REGION Network 41: RO-2 A AUTO FLUSING VALVE AGLV-401 CLOSE COMMOND FAIL
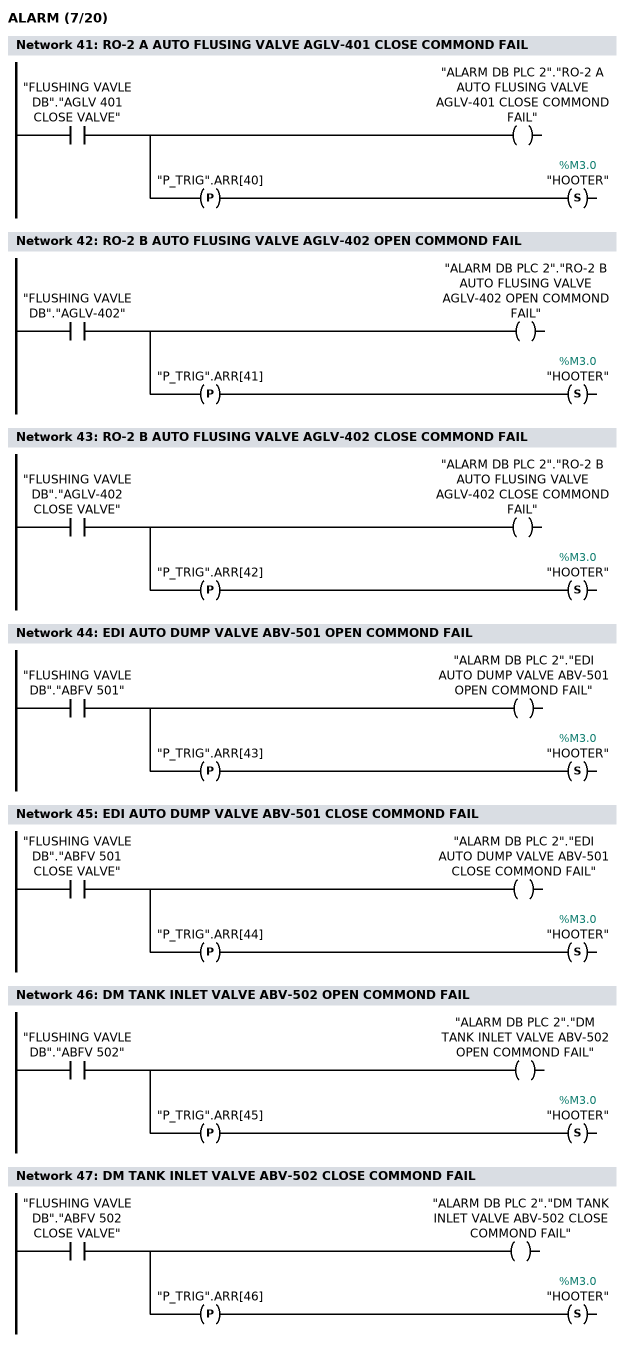
   RUNG wire#powerrail
      Contact( "FLUSHING VAVLE DB"."AGLV 401 CLOSE VALVE" )
      wire#w1
      Coil( "ALARM DB PLC 2"."RO-2 A AUTO FLUSING VALVE AGLV-401 CLOSE COMMOND FAIL" )
   END_RUNG
   RUNG wire#w1
      P_Trig( "P_TRIG".ARR[40] )
      S_Coil( "HOOTER" )
   END_RUNG
   // the same network as SCL:
   "ALARM DB PLC 2"."RO-2 A AUTO FLUSING VALVE AGLV-401 CLOSE COMMOND FAIL" := "FLUSHING VAVLE DB"."AGLV 401 CLOSE VALVE";
   #_w1 := "FLUSHING VAVLE DB"."AGLV 401 CLOSE VALVE" AND NOT "P_TRIG".ARR[40];   // rising edge
   "P_TRIG".ARR[40] := "FLUSHING VAVLE DB"."AGLV 401 CLOSE VALVE";
   IF #_w1 THEN "HOOTER" := TRUE; END_IF;
END_REGION

REGION Network 42: RO-2 B AUTO FLUSING VALVE AGLV-402 OPEN COMMOND FAIL
   RUNG wire#powerrail
      Contact( "FLUSHING VAVLE DB"."AGLV-402" )
      wire#w1
      Coil( "ALARM DB PLC 2"."RO-2 B AUTO FLUSING VALVE AGLV-402 OPEN COMMOND FAIL" )
   END_RUNG
   RUNG wire#w1
      P_Trig( "P_TRIG".ARR[41] )
      S_Coil( "HOOTER" )
   END_RUNG
   // the same network as SCL:
   "ALARM DB PLC 2"."RO-2 B AUTO FLUSING VALVE AGLV-402 OPEN COMMOND FAIL" := "FLUSHING VAVLE DB"."AGLV-402";
   #_w1 := "FLUSHING VAVLE DB"."AGLV-402" AND NOT "P_TRIG".ARR[41];   // rising edge
   "P_TRIG".ARR[41] := "FLUSHING VAVLE DB"."AGLV-402";
   IF #_w1 THEN "HOOTER" := TRUE; END_IF;
END_REGION

REGION Network 43: RO-2 B AUTO FLUSING VALVE AGLV-402 CLOSE COMMOND FAIL
   RUNG wire#powerrail
      Contact( "FLUSHING VAVLE DB"."AGLV-402 CLOSE VALVE" )
      wire#w1
      Coil( "ALARM DB PLC 2"."RO-2 B AUTO FLUSING VALVE AGLV-402 CLOSE COMMOND FAIL" )
   END_RUNG
   RUNG wire#w1
      P_Trig( "P_TRIG".ARR[42] )
      S_Coil( "HOOTER" )
   END_RUNG
   // the same network as SCL:
   "ALARM DB PLC 2"."RO-2 B AUTO FLUSING VALVE AGLV-402 CLOSE COMMOND FAIL" := "FLUSHING VAVLE DB"."AGLV-402 CLOSE VALVE";
   #_w1 := "FLUSHING VAVLE DB"."AGLV-402 CLOSE VALVE" AND NOT "P_TRIG".ARR[42];   // rising edge
   "P_TRIG".ARR[42] := "FLUSHING VAVLE DB"."AGLV-402 CLOSE VALVE";
   IF #_w1 THEN "HOOTER" := TRUE; END_IF;
END_REGION

REGION Network 44: EDI AUTO DUMP VALVE ABV-501 OPEN COMMOND FAIL
   RUNG wire#powerrail
      Contact( "FLUSHING VAVLE DB"."ABFV 501" )
      wire#w1
      Coil( "ALARM DB PLC 2"."EDI AUTO DUMP VALVE ABV-501 OPEN COMMOND FAIL" )
   END_RUNG
   RUNG wire#w1
      P_Trig( "P_TRIG".ARR[43] )
      S_Coil( "HOOTER" )
   END_RUNG
   // the same network as SCL:
   "ALARM DB PLC 2"."EDI AUTO DUMP VALVE ABV-501 OPEN COMMOND FAIL" := "FLUSHING VAVLE DB"."ABFV 501";
   #_w1 := "FLUSHING VAVLE DB"."ABFV 501" AND NOT "P_TRIG".ARR[43];   // rising edge
   "P_TRIG".ARR[43] := "FLUSHING VAVLE DB"."ABFV 501";
   IF #_w1 THEN "HOOTER" := TRUE; END_IF;
END_REGION

REGION Network 45: EDI AUTO DUMP VALVE ABV-501 CLOSE COMMOND FAIL
   RUNG wire#powerrail
      Contact( "FLUSHING VAVLE DB"."ABFV 501 CLOSE VALVE" )
      wire#w1
      Coil( "ALARM DB PLC 2"."EDI AUTO DUMP VALVE ABV-501 CLOSE COMMOND FAIL" )
   END_RUNG
   RUNG wire#w1
      P_Trig( "P_TRIG".ARR[44] )
      S_Coil( "HOOTER" )
   END_RUNG
   // the same network as SCL:
   "ALARM DB PLC 2"."EDI AUTO DUMP VALVE ABV-501 CLOSE COMMOND FAIL" := "FLUSHING VAVLE DB"."ABFV 501 CLOSE VALVE";
   #_w1 := "FLUSHING VAVLE DB"."ABFV 501 CLOSE VALVE" AND NOT "P_TRIG".ARR[44];   // rising edge
   "P_TRIG".ARR[44] := "FLUSHING VAVLE DB"."ABFV 501 CLOSE VALVE";
   IF #_w1 THEN "HOOTER" := TRUE; END_IF;
END_REGION

REGION Network 46: DM TANK INLET VALVE ABV-502 OPEN COMMOND FAIL
   RUNG wire#powerrail
      Contact( "FLUSHING VAVLE DB"."ABFV 502" )
      wire#w1
      Coil( "ALARM DB PLC 2"."DM TANK INLET VALVE ABV-502 OPEN COMMOND FAIL" )
   END_RUNG
   RUNG wire#w1
      P_Trig( "P_TRIG".ARR[45] )
      S_Coil( "HOOTER" )
   END_RUNG
   // the same network as SCL:
   "ALARM DB PLC 2"."DM TANK INLET VALVE ABV-502 OPEN COMMOND FAIL" := "FLUSHING VAVLE DB"."ABFV 502";
   #_w1 := "FLUSHING VAVLE DB"."ABFV 502" AND NOT "P_TRIG".ARR[45];   // rising edge
   "P_TRIG".ARR[45] := "FLUSHING VAVLE DB"."ABFV 502";
   IF #_w1 THEN "HOOTER" := TRUE; END_IF;
END_REGION

REGION Network 47: DM TANK INLET VALVE ABV-502 CLOSE COMMOND FAIL
   RUNG wire#powerrail
      Contact( "FLUSHING VAVLE DB"."ABFV 502 CLOSE VALVE" )
      wire#w1
      Coil( "ALARM DB PLC 2"."DM TANK INLET VALVE ABV-502 CLOSE COMMOND FAIL" )
   END_RUNG
   RUNG wire#w1
      P_Trig( "P_TRIG".ARR[46] )
      S_Coil( "HOOTER" )
   END_RUNG
   // the same network as SCL:
   "ALARM DB PLC 2"."DM TANK INLET VALVE ABV-502 CLOSE COMMOND FAIL" := "FLUSHING VAVLE DB"."ABFV 502 CLOSE VALVE";
   #_w1 := "FLUSHING VAVLE DB"."ABFV 502 CLOSE VALVE" AND NOT "P_TRIG".ARR[46];   // rising edge
   "P_TRIG".ARR[46] := "FLUSHING VAVLE DB"."ABFV 502 CLOSE VALVE";
   IF #_w1 THEN "HOOTER" := TRUE; END_IF;
END_REGION

REGION Network 48: RO-02 FEED TANK LEVEL ( LT-401)- LOW LOW
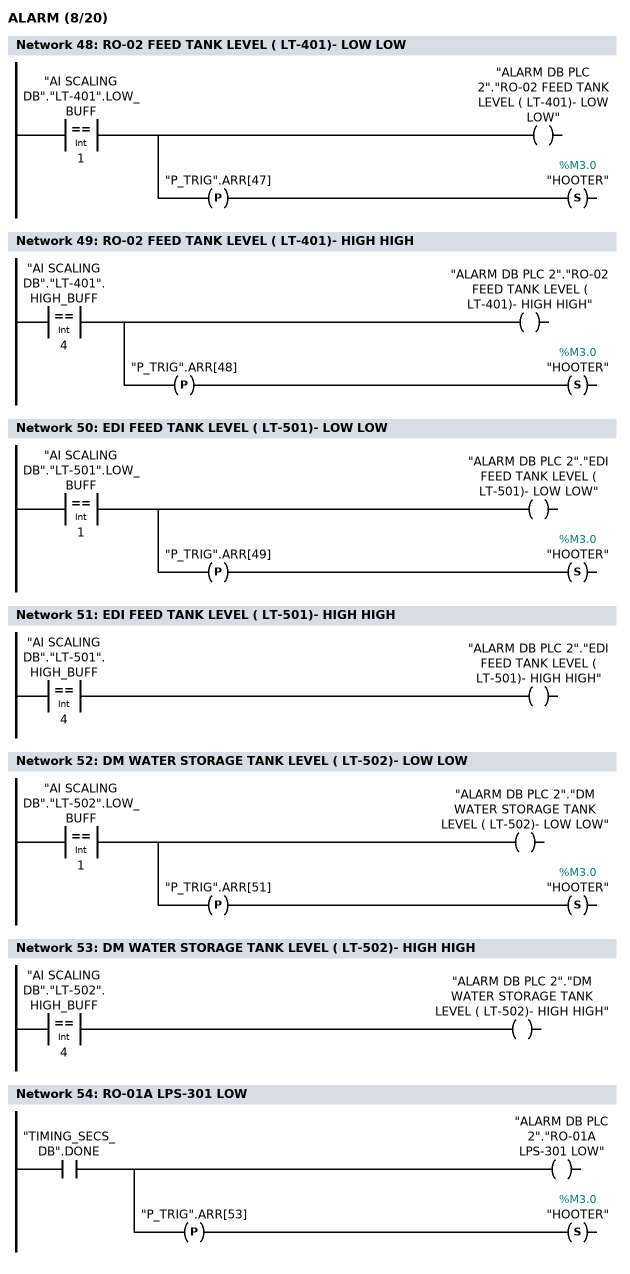
   RUNG wire#powerrail
      { S7_Templates := "SrcType := Int" } EQ_Contact(in1 := "AI SCALING DB"."LT-401".LOW_BUFF, in2 := 1)
      wire#w1
      Coil( "ALARM DB PLC 2"."RO-02 FEED TANK LEVEL ( LT-401)- LOW LOW" )
   END_RUNG
   RUNG wire#w1
      P_Trig( "P_TRIG".ARR[47] )
      S_Coil( "HOOTER" )
   END_RUNG
   // the same network as SCL:
   "ALARM DB PLC 2"."RO-02 FEED TANK LEVEL ( LT-401)- LOW LOW" := "AI SCALING DB"."LT-401".LOW_BUFF = 1;
   #_w1 := "ALARM DB PLC 2"."RO-02 FEED TANK LEVEL ( LT-401)- LOW LOW" AND NOT "P_TRIG".ARR[47];   // rising edge
   "P_TRIG".ARR[47] := "ALARM DB PLC 2"."RO-02 FEED TANK LEVEL ( LT-401)- LOW LOW";
   IF #_w1 THEN "HOOTER" := TRUE; END_IF;
END_REGION

REGION Network 49: RO-02 FEED TANK LEVEL ( LT-401)- HIGH HIGH
   RUNG wire#powerrail
      { S7_Templates := "SrcType := Int" } EQ_Contact(in1 := "AI SCALING DB"."LT-401".HIGH_BUFF, in2 := 4)
      wire#w1
      Coil( "ALARM DB PLC 2"."RO-02 FEED TANK LEVEL ( LT-401)- HIGH HIGH" )
   END_RUNG
   RUNG wire#w1
      P_Trig( "P_TRIG".ARR[48] )
      S_Coil( "HOOTER" )
   END_RUNG
   // the same network as SCL:
   "ALARM DB PLC 2"."RO-02 FEED TANK LEVEL ( LT-401)- HIGH HIGH" := "AI SCALING DB"."LT-401".HIGH_BUFF = 4;
   #_w1 := "ALARM DB PLC 2"."RO-02 FEED TANK LEVEL ( LT-401)- HIGH HIGH" AND NOT "P_TRIG".ARR[48];   // rising edge
   "P_TRIG".ARR[48] := "ALARM DB PLC 2"."RO-02 FEED TANK LEVEL ( LT-401)- HIGH HIGH";
   IF #_w1 THEN "HOOTER" := TRUE; END_IF;
END_REGION

REGION Network 50: EDI FEED TANK LEVEL ( LT-501)- LOW LOW
   RUNG wire#powerrail
      { S7_Templates := "SrcType := Int" } EQ_Contact(in1 := "AI SCALING DB"."LT-501".LOW_BUFF, in2 := 1)
      wire#w1
      Coil( "ALARM DB PLC 2"."EDI FEED TANK LEVEL ( LT-501)- LOW LOW" )
   END_RUNG
   RUNG wire#w1
      P_Trig( "P_TRIG".ARR[49] )
      S_Coil( "HOOTER" )
   END_RUNG
   // the same network as SCL:
   "ALARM DB PLC 2"."EDI FEED TANK LEVEL ( LT-501)- LOW LOW" := "AI SCALING DB"."LT-501".LOW_BUFF = 1;
   #_w1 := "ALARM DB PLC 2"."EDI FEED TANK LEVEL ( LT-501)- LOW LOW" AND NOT "P_TRIG".ARR[49];   // rising edge
   "P_TRIG".ARR[49] := "ALARM DB PLC 2"."EDI FEED TANK LEVEL ( LT-501)- LOW LOW";
   IF #_w1 THEN "HOOTER" := TRUE; END_IF;
END_REGION

REGION Network 51: EDI FEED TANK LEVEL ( LT-501)- HIGH HIGH
   RUNG wire#powerrail
      { S7_Templates := "SrcType := Int" } EQ_Contact(in1 := "AI SCALING DB"."LT-501".HIGH_BUFF, in2 := 4)
      Coil( "ALARM DB PLC 2"."EDI FEED TANK LEVEL ( LT-501)- HIGH HIGH" )
   END_RUNG
   // the same network as SCL:
   "ALARM DB PLC 2"."EDI FEED TANK LEVEL ( LT-501)- HIGH HIGH" := "AI SCALING DB"."LT-501".HIGH_BUFF = 4;
END_REGION

REGION Network 52: DM WATER STORAGE TANK LEVEL ( LT-502)- LOW LOW
   RUNG wire#powerrail
      { S7_Templates := "SrcType := Int" } EQ_Contact(in1 := "AI SCALING DB"."LT-502".LOW_BUFF, in2 := 1)
      wire#w1
      Coil( "ALARM DB PLC 2"."DM WATER STORAGE TANK  LEVEL ( LT-502)- LOW LOW" )
   END_RUNG
   RUNG wire#w1
      P_Trig( "P_TRIG".ARR[51] )
      S_Coil( "HOOTER" )
   END_RUNG
   // the same network as SCL:
   "ALARM DB PLC 2"."DM WATER STORAGE TANK  LEVEL ( LT-502)- LOW LOW" := "AI SCALING DB"."LT-502".LOW_BUFF = 1;
   #_w1 := "ALARM DB PLC 2"."DM WATER STORAGE TANK  LEVEL ( LT-502)- LOW LOW" AND NOT "P_TRIG".ARR[51];   // rising edge
   "P_TRIG".ARR[51] := "ALARM DB PLC 2"."DM WATER STORAGE TANK  LEVEL ( LT-502)- LOW LOW";
   IF #_w1 THEN "HOOTER" := TRUE; END_IF;
END_REGION

REGION Network 53: DM WATER STORAGE TANK LEVEL ( LT-502)- HIGH HIGH
   RUNG wire#powerrail
      { S7_Templates := "SrcType := Int" } EQ_Contact(in1 := "AI SCALING DB"."LT-502".HIGH_BUFF, in2 := 4)
      Coil( "ALARM DB PLC 2"."DM WATER STORAGE TANK LEVEL ( LT-502)- HIGH HIGH" )
   END_RUNG
   // the same network as SCL:
   "ALARM DB PLC 2"."DM WATER STORAGE TANK LEVEL ( LT-502)- HIGH HIGH" := "AI SCALING DB"."LT-502".HIGH_BUFF = 4;
END_REGION

REGION Network 54: RO-01A LPS-301 LOW
   RUNG wire#powerrail
      Contact( "TIMING_SECS_DB".DONE )
      wire#w1
      Coil( "ALARM DB PLC 2"."RO-01A LPS-301 LOW" )
   END_RUNG
   RUNG wire#w1
      P_Trig( "P_TRIG".ARR[53] )
      S_Coil( "HOOTER" )
   END_RUNG
   // the same network as SCL:
   "ALARM DB PLC 2"."RO-01A LPS-301 LOW" := "TIMING_SECS_DB".DONE;
   #_w1 := "TIMING_SECS_DB".DONE AND NOT "P_TRIG".ARR[53];   // rising edge
   "P_TRIG".ARR[53] := "TIMING_SECS_DB".DONE;
   IF #_w1 THEN "HOOTER" := TRUE; END_IF;
END_REGION

REGION Network 55: RO-01 B LPS-302 LOW
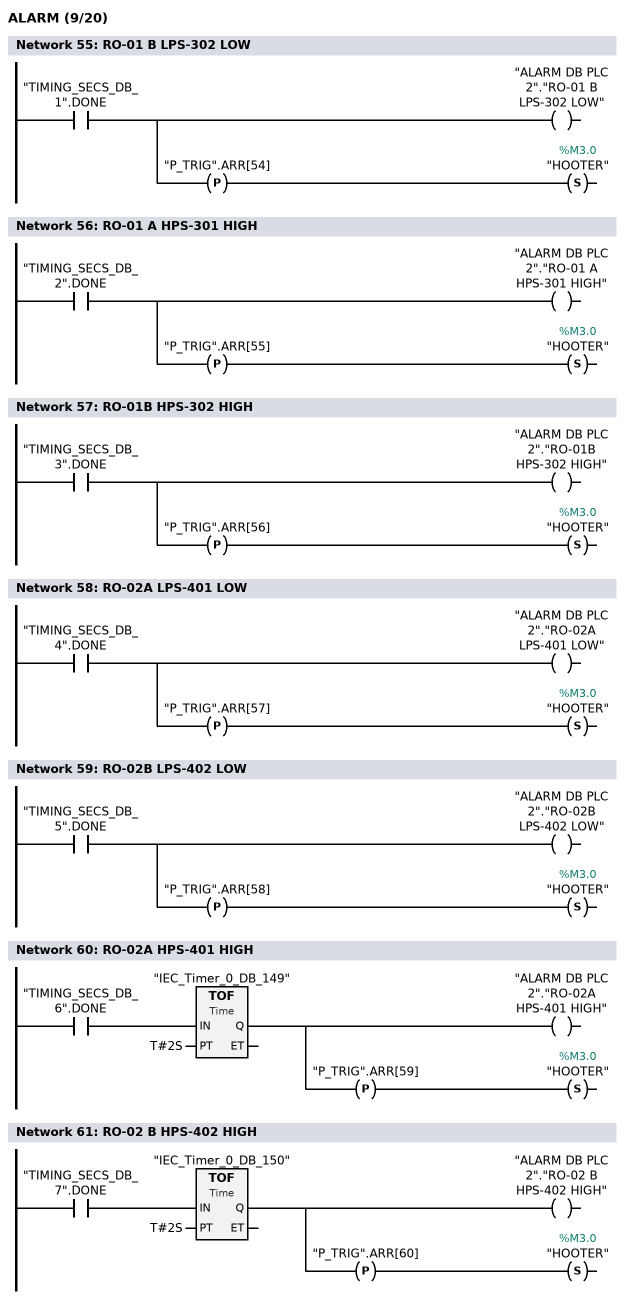
   RUNG wire#powerrail
      Contact( "TIMING_SECS_DB_1".DONE )
      wire#w1
      Coil( "ALARM DB PLC 2"."RO-01 B LPS-302 LOW" )
   END_RUNG
   RUNG wire#w1
      P_Trig( "P_TRIG".ARR[54] )
      S_Coil( "HOOTER" )
   END_RUNG
   // the same network as SCL:
   "ALARM DB PLC 2"."RO-01 B LPS-302 LOW" := "TIMING_SECS_DB_1".DONE;
   #_w1 := "TIMING_SECS_DB_1".DONE AND NOT "P_TRIG".ARR[54];   // rising edge
   "P_TRIG".ARR[54] := "TIMING_SECS_DB_1".DONE;
   IF #_w1 THEN "HOOTER" := TRUE; END_IF;
END_REGION

REGION Network 56: RO-01 A HPS-301 HIGH
   RUNG wire#powerrail
      Contact( "TIMING_SECS_DB_2".DONE )
      wire#w1
      Coil( "ALARM DB PLC 2"."RO-01 A HPS-301 HIGH" )
   END_RUNG
   RUNG wire#w1
      P_Trig( "P_TRIG".ARR[55] )
      S_Coil( "HOOTER" )
   END_RUNG
   // the same network as SCL:
   "ALARM DB PLC 2"."RO-01 A HPS-301 HIGH" := "TIMING_SECS_DB_2".DONE;
   #_w1 := "TIMING_SECS_DB_2".DONE AND NOT "P_TRIG".ARR[55];   // rising edge
   "P_TRIG".ARR[55] := "TIMING_SECS_DB_2".DONE;
   IF #_w1 THEN "HOOTER" := TRUE; END_IF;
END_REGION

REGION Network 57: RO-01B HPS-302 HIGH
   RUNG wire#powerrail
      Contact( "TIMING_SECS_DB_3".DONE )
      wire#w1
      Coil( "ALARM DB PLC 2"."RO-01B HPS-302 HIGH" )
   END_RUNG
   RUNG wire#w1
      P_Trig( "P_TRIG".ARR[56] )
      S_Coil( "HOOTER" )
   END_RUNG
   // the same network as SCL:
   "ALARM DB PLC 2"."RO-01B HPS-302 HIGH" := "TIMING_SECS_DB_3".DONE;
   #_w1 := "TIMING_SECS_DB_3".DONE AND NOT "P_TRIG".ARR[56];   // rising edge
   "P_TRIG".ARR[56] := "TIMING_SECS_DB_3".DONE;
   IF #_w1 THEN "HOOTER" := TRUE; END_IF;
END_REGION

REGION Network 58: RO-02A LPS-401 LOW
   RUNG wire#powerrail
      Contact( "TIMING_SECS_DB_4".DONE )
      wire#w1
      Coil( "ALARM DB PLC 2"."RO-02A LPS-401 LOW" )
   END_RUNG
   RUNG wire#w1
      P_Trig( "P_TRIG".ARR[57] )
      S_Coil( "HOOTER" )
   END_RUNG
   // the same network as SCL:
   "ALARM DB PLC 2"."RO-02A LPS-401 LOW" := "TIMING_SECS_DB_4".DONE;
   #_w1 := "TIMING_SECS_DB_4".DONE AND NOT "P_TRIG".ARR[57];   // rising edge
   "P_TRIG".ARR[57] := "TIMING_SECS_DB_4".DONE;
   IF #_w1 THEN "HOOTER" := TRUE; END_IF;
END_REGION

REGION Network 59: RO-02B LPS-402 LOW
   RUNG wire#powerrail
      Contact( "TIMING_SECS_DB_5".DONE )
      wire#w1
      Coil( "ALARM DB PLC 2"."RO-02B LPS-402 LOW" )
   END_RUNG
   RUNG wire#w1
      P_Trig( "P_TRIG".ARR[58] )
      S_Coil( "HOOTER" )
   END_RUNG
   // the same network as SCL:
   "ALARM DB PLC 2"."RO-02B LPS-402 LOW" := "TIMING_SECS_DB_5".DONE;
   #_w1 := "TIMING_SECS_DB_5".DONE AND NOT "P_TRIG".ARR[58];   // rising edge
   "P_TRIG".ARR[58] := "TIMING_SECS_DB_5".DONE;
   IF #_w1 THEN "HOOTER" := TRUE; END_IF;
END_REGION

REGION Network 60: RO-02A HPS-401 HIGH
   RUNG wire#powerrail
      Contact( "TIMING_SECS_DB_6".DONE )
      { S7_Templates := "time_type := Time" } "IEC_Timer_0_DB_149".TOF(pt := T#2S, et =>)
      wire#w1
      Coil( "ALARM DB PLC 2"."RO-02A HPS-401 HIGH" )
   END_RUNG
   RUNG wire#w1
      P_Trig( "P_TRIG".ARR[59] )
      S_Coil( "HOOTER" )
   END_RUNG
   // the same network as SCL:
   "IEC_Timer_0_DB_149".TOF(IN := "TIMING_SECS_DB_6".DONE, PT := T#2S);
   "ALARM DB PLC 2"."RO-02A HPS-401 HIGH" := "IEC_Timer_0_DB_149".Q;
   #_w1 := "IEC_Timer_0_DB_149".Q AND NOT "P_TRIG".ARR[59];   // rising edge
   "P_TRIG".ARR[59] := "IEC_Timer_0_DB_149".Q;
   IF #_w1 THEN "HOOTER" := TRUE; END_IF;
END_REGION

REGION Network 61: RO-02 B HPS-402 HIGH
   RUNG wire#powerrail
      Contact( "TIMING_SECS_DB_7".DONE )
      { S7_Templates := "time_type := Time" } "IEC_Timer_0_DB_150".TOF(pt := T#2S, et =>)
      wire#w1
      Coil( "ALARM DB PLC 2"."RO-02 B HPS-402 HIGH" )
   END_RUNG
   RUNG wire#w1
      P_Trig( "P_TRIG".ARR[60] )
      S_Coil( "HOOTER" )
   END_RUNG
   // the same network as SCL:
   "IEC_Timer_0_DB_150".TOF(IN := "TIMING_SECS_DB_7".DONE, PT := T#2S);
   "ALARM DB PLC 2"."RO-02 B HPS-402 HIGH" := "IEC_Timer_0_DB_150".Q;
   #_w1 := "IEC_Timer_0_DB_150".Q AND NOT "P_TRIG".ARR[60];   // rising edge
   "P_TRIG".ARR[60] := "IEC_Timer_0_DB_150".Q;
   IF #_w1 THEN "HOOTER" := TRUE; END_IF;
END_REGION

REGION Network 62: EDI-501A FEED PRESSURE PT-501 LOW
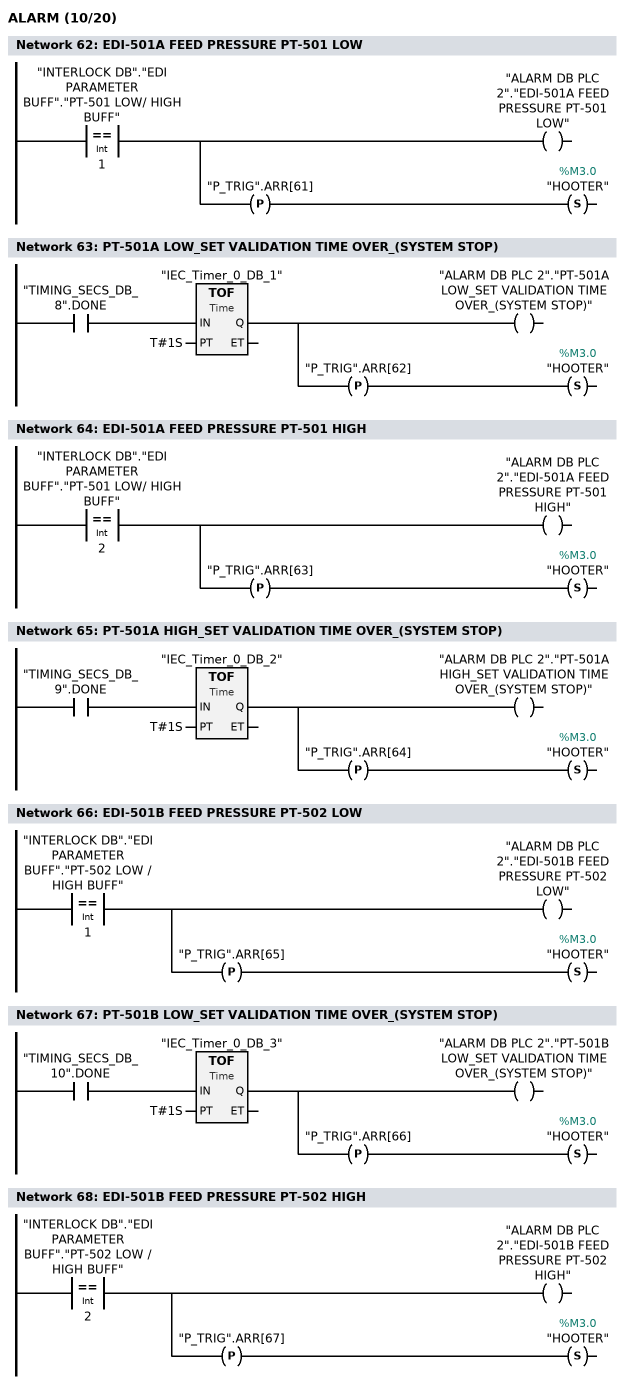
   RUNG wire#powerrail
      { S7_Templates := "SrcType := Int" } EQ_Contact(in1 := "INTERLOCK DB"."EDI PARAMETER BUFF"."PT-501 LOW/ HIGH BUFF", in2 := 1)
      wire#w1
      Coil( "ALARM DB PLC 2"."EDI-501A FEED PRESSURE PT-501 LOW" )
   END_RUNG
   RUNG wire#w1
      P_Trig( "P_TRIG".ARR[61] )
      S_Coil( "HOOTER" )
   END_RUNG
   // the same network as SCL:
   "ALARM DB PLC 2"."EDI-501A FEED PRESSURE PT-501 LOW" := "INTERLOCK DB"."EDI PARAMETER BUFF"."PT-501 LOW/ HIGH BUFF" = 1;
   #_w1 := "ALARM DB PLC 2"."EDI-501A FEED PRESSURE PT-501 LOW" AND NOT "P_TRIG".ARR[61];   // rising edge
   "P_TRIG".ARR[61] := "ALARM DB PLC 2"."EDI-501A FEED PRESSURE PT-501 LOW";
   IF #_w1 THEN "HOOTER" := TRUE; END_IF;
END_REGION

REGION Network 63: PT-501A LOW_SET VALIDATION TIME OVER_(SYSTEM STOP)
   RUNG wire#powerrail
      Contact( "TIMING_SECS_DB_8".DONE )
      { S7_Templates := "time_type := Time" } "IEC_Timer_0_DB_1".TOF(pt := T#1S, et =>)
      wire#w1
      Coil( "ALARM DB PLC 2"."PT-501A LOW_SET VALIDATION TIME OVER_(SYSTEM STOP)" )
   END_RUNG
   RUNG wire#w1
      P_Trig( "P_TRIG".ARR[62] )
      S_Coil( "HOOTER" )
   END_RUNG
   // the same network as SCL:
   "IEC_Timer_0_DB_1".TOF(IN := "TIMING_SECS_DB_8".DONE, PT := T#1S);
   "ALARM DB PLC 2"."PT-501A LOW_SET VALIDATION TIME OVER_(SYSTEM STOP)" := "IEC_Timer_0_DB_1".Q;
   #_w1 := "IEC_Timer_0_DB_1".Q AND NOT "P_TRIG".ARR[62];   // rising edge
   "P_TRIG".ARR[62] := "IEC_Timer_0_DB_1".Q;
   IF #_w1 THEN "HOOTER" := TRUE; END_IF;
END_REGION

REGION Network 64: EDI-501A FEED PRESSURE PT-501 HIGH
   RUNG wire#powerrail
      { S7_Templates := "SrcType := Int" } EQ_Contact(in1 := "INTERLOCK DB"."EDI PARAMETER BUFF"."PT-501 LOW/ HIGH BUFF", in2 := 2)
      wire#w1
      Coil( "ALARM DB PLC 2"."EDI-501A FEED PRESSURE PT-501 HIGH" )
   END_RUNG
   RUNG wire#w1
      P_Trig( "P_TRIG".ARR[63] )
      S_Coil( "HOOTER" )
   END_RUNG
   // the same network as SCL:
   "ALARM DB PLC 2"."EDI-501A FEED PRESSURE PT-501 HIGH" := "INTERLOCK DB"."EDI PARAMETER BUFF"."PT-501 LOW/ HIGH BUFF" = 2;
   #_w1 := "ALARM DB PLC 2"."EDI-501A FEED PRESSURE PT-501 HIGH" AND NOT "P_TRIG".ARR[63];   // rising edge
   "P_TRIG".ARR[63] := "ALARM DB PLC 2"."EDI-501A FEED PRESSURE PT-501 HIGH";
   IF #_w1 THEN "HOOTER" := TRUE; END_IF;
END_REGION

REGION Network 65: PT-501A HIGH_SET VALIDATION TIME OVER_(SYSTEM STOP)
   RUNG wire#powerrail
      Contact( "TIMING_SECS_DB_9".DONE )
      { S7_Templates := "time_type := Time" } "IEC_Timer_0_DB_2".TOF(pt := T#1S, et =>)
      wire#w1
      Coil( "ALARM DB PLC 2"."PT-501A HIGH_SET VALIDATION TIME OVER_(SYSTEM STOP)" )
   END_RUNG
   RUNG wire#w1
      P_Trig( "P_TRIG".ARR[64] )
      S_Coil( "HOOTER" )
   END_RUNG
   // the same network as SCL:
   "IEC_Timer_0_DB_2".TOF(IN := "TIMING_SECS_DB_9".DONE, PT := T#1S);
   "ALARM DB PLC 2"."PT-501A HIGH_SET VALIDATION TIME OVER_(SYSTEM STOP)" := "IEC_Timer_0_DB_2".Q;
   #_w1 := "IEC_Timer_0_DB_2".Q AND NOT "P_TRIG".ARR[64];   // rising edge
   "P_TRIG".ARR[64] := "IEC_Timer_0_DB_2".Q;
   IF #_w1 THEN "HOOTER" := TRUE; END_IF;
END_REGION

REGION Network 66: EDI-501B FEED PRESSURE PT-502 LOW
   RUNG wire#powerrail
      { S7_Templates := "SrcType := Int" } EQ_Contact(in1 := "INTERLOCK DB"."EDI PARAMETER BUFF"."PT-502 LOW / HIGH BUFF", in2 := 1)
      wire#w1
      Coil( "ALARM DB PLC 2"."EDI-501B FEED PRESSURE PT-502 LOW" )
   END_RUNG
   RUNG wire#w1
      P_Trig( "P_TRIG".ARR[65] )
      S_Coil( "HOOTER" )
   END_RUNG
   // the same network as SCL:
   "ALARM DB PLC 2"."EDI-501B FEED PRESSURE PT-502 LOW" := "INTERLOCK DB"."EDI PARAMETER BUFF"."PT-502 LOW / HIGH BUFF" = 1;
   #_w1 := "ALARM DB PLC 2"."EDI-501B FEED PRESSURE PT-502 LOW" AND NOT "P_TRIG".ARR[65];   // rising edge
   "P_TRIG".ARR[65] := "ALARM DB PLC 2"."EDI-501B FEED PRESSURE PT-502 LOW";
   IF #_w1 THEN "HOOTER" := TRUE; END_IF;
END_REGION

REGION Network 67: PT-501B LOW_SET VALIDATION TIME OVER_(SYSTEM STOP)
   RUNG wire#powerrail
      Contact( "TIMING_SECS_DB_10".DONE )
      { S7_Templates := "time_type := Time" } "IEC_Timer_0_DB_3".TOF(pt := T#1S, et =>)
      wire#w1
      Coil( "ALARM DB PLC 2"."PT-501B LOW_SET VALIDATION TIME OVER_(SYSTEM STOP)" )
   END_RUNG
   RUNG wire#w1
      P_Trig( "P_TRIG".ARR[66] )
      S_Coil( "HOOTER" )
   END_RUNG
   // the same network as SCL:
   "IEC_Timer_0_DB_3".TOF(IN := "TIMING_SECS_DB_10".DONE, PT := T#1S);
   "ALARM DB PLC 2"."PT-501B LOW_SET VALIDATION TIME OVER_(SYSTEM STOP)" := "IEC_Timer_0_DB_3".Q;
   #_w1 := "IEC_Timer_0_DB_3".Q AND NOT "P_TRIG".ARR[66];   // rising edge
   "P_TRIG".ARR[66] := "IEC_Timer_0_DB_3".Q;
   IF #_w1 THEN "HOOTER" := TRUE; END_IF;
END_REGION

REGION Network 68: EDI-501B FEED PRESSURE PT-502 HIGH
   RUNG wire#powerrail
      { S7_Templates := "SrcType := Int" } EQ_Contact(in1 := "INTERLOCK DB"."EDI PARAMETER BUFF"."PT-502 LOW / HIGH BUFF", in2 := 2)
      wire#w1
      Coil( "ALARM DB PLC 2"."EDI-501B FEED PRESSURE PT-502 HIGH" )
   END_RUNG
   RUNG wire#w1
      P_Trig( "P_TRIG".ARR[67] )
      S_Coil( "HOOTER" )
   END_RUNG
   // the same network as SCL:
   "ALARM DB PLC 2"."EDI-501B FEED PRESSURE PT-502 HIGH" := "INTERLOCK DB"."EDI PARAMETER BUFF"."PT-502 LOW / HIGH BUFF" = 2;
   #_w1 := "ALARM DB PLC 2"."EDI-501B FEED PRESSURE PT-502 HIGH" AND NOT "P_TRIG".ARR[67];   // rising edge
   "P_TRIG".ARR[67] := "ALARM DB PLC 2"."EDI-501B FEED PRESSURE PT-502 HIGH";
   IF #_w1 THEN "HOOTER" := TRUE; END_IF;
END_REGION

REGION Network 69: PT-501B HIGH_SET VALIDATION TIME OVER_(SYSTEM STOP)
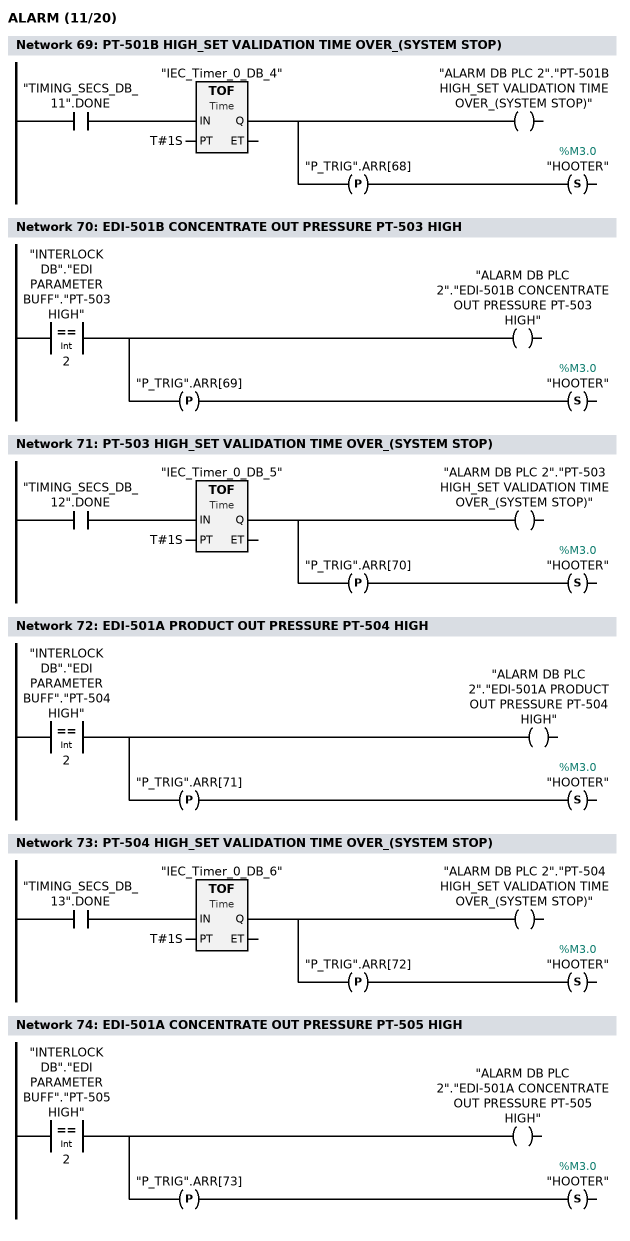
   RUNG wire#powerrail
      Contact( "TIMING_SECS_DB_11".DONE )
      { S7_Templates := "time_type := Time" } "IEC_Timer_0_DB_4".TOF(pt := T#1S, et =>)
      wire#w1
      Coil( "ALARM DB PLC 2"."PT-501B HIGH_SET VALIDATION TIME OVER_(SYSTEM STOP)" )
   END_RUNG
   RUNG wire#w1
      P_Trig( "P_TRIG".ARR[68] )
      S_Coil( "HOOTER" )
   END_RUNG
   // the same network as SCL:
   "IEC_Timer_0_DB_4".TOF(IN := "TIMING_SECS_DB_11".DONE, PT := T#1S);
   "ALARM DB PLC 2"."PT-501B HIGH_SET VALIDATION TIME OVER_(SYSTEM STOP)" := "IEC_Timer_0_DB_4".Q;
   #_w1 := "IEC_Timer_0_DB_4".Q AND NOT "P_TRIG".ARR[68];   // rising edge
   "P_TRIG".ARR[68] := "IEC_Timer_0_DB_4".Q;
   IF #_w1 THEN "HOOTER" := TRUE; END_IF;
END_REGION

REGION Network 70: EDI-501B CONCENTRATE OUT PRESSURE PT-503 HIGH
   RUNG wire#powerrail
      { S7_Templates := "SrcType := Int" } EQ_Contact(in1 := "INTERLOCK DB"."EDI PARAMETER BUFF"."PT-503 HIGH", in2 := 2)
      wire#w1
      Coil( "ALARM DB PLC 2"."EDI-501B CONCENTRATE OUT PRESSURE PT-503 HIGH" )
   END_RUNG
   RUNG wire#w1
      P_Trig( "P_TRIG".ARR[69] )
      S_Coil( "HOOTER" )
   END_RUNG
   // the same network as SCL:
   "ALARM DB PLC 2"."EDI-501B CONCENTRATE OUT PRESSURE PT-503 HIGH" := "INTERLOCK DB"."EDI PARAMETER BUFF"."PT-503 HIGH" = 2;
   #_w1 := "ALARM DB PLC 2"."EDI-501B CONCENTRATE OUT PRESSURE PT-503 HIGH" AND NOT "P_TRIG".ARR[69];   // rising edge
   "P_TRIG".ARR[69] := "ALARM DB PLC 2"."EDI-501B CONCENTRATE OUT PRESSURE PT-503 HIGH";
   IF #_w1 THEN "HOOTER" := TRUE; END_IF;
END_REGION

REGION Network 71: PT-503 HIGH_SET VALIDATION TIME OVER_(SYSTEM STOP)
   RUNG wire#powerrail
      Contact( "TIMING_SECS_DB_12".DONE )
      { S7_Templates := "time_type := Time" } "IEC_Timer_0_DB_5".TOF(pt := T#1S, et =>)
      wire#w1
      Coil( "ALARM DB PLC 2"."PT-503 HIGH_SET VALIDATION TIME OVER_(SYSTEM STOP)" )
   END_RUNG
   RUNG wire#w1
      P_Trig( "P_TRIG".ARR[70] )
      S_Coil( "HOOTER" )
   END_RUNG
   // the same network as SCL:
   "IEC_Timer_0_DB_5".TOF(IN := "TIMING_SECS_DB_12".DONE, PT := T#1S);
   "ALARM DB PLC 2"."PT-503 HIGH_SET VALIDATION TIME OVER_(SYSTEM STOP)" := "IEC_Timer_0_DB_5".Q;
   #_w1 := "IEC_Timer_0_DB_5".Q AND NOT "P_TRIG".ARR[70];   // rising edge
   "P_TRIG".ARR[70] := "IEC_Timer_0_DB_5".Q;
   IF #_w1 THEN "HOOTER" := TRUE; END_IF;
END_REGION

REGION Network 72: EDI-501A PRODUCT OUT PRESSURE PT-504 HIGH
   RUNG wire#powerrail
      { S7_Templates := "SrcType := Int" } EQ_Contact(in1 := "INTERLOCK DB"."EDI PARAMETER BUFF"."PT-504 HIGH", in2 := 2)
      wire#w1
      Coil( "ALARM DB PLC 2"."EDI-501A PRODUCT OUT PRESSURE PT-504 HIGH" )
   END_RUNG
   RUNG wire#w1
      P_Trig( "P_TRIG".ARR[71] )
      S_Coil( "HOOTER" )
   END_RUNG
   // the same network as SCL:
   "ALARM DB PLC 2"."EDI-501A PRODUCT OUT PRESSURE PT-504 HIGH" := "INTERLOCK DB"."EDI PARAMETER BUFF"."PT-504 HIGH" = 2;
   #_w1 := "ALARM DB PLC 2"."EDI-501A PRODUCT OUT PRESSURE PT-504 HIGH" AND NOT "P_TRIG".ARR[71];   // rising edge
   "P_TRIG".ARR[71] := "ALARM DB PLC 2"."EDI-501A PRODUCT OUT PRESSURE PT-504 HIGH";
   IF #_w1 THEN "HOOTER" := TRUE; END_IF;
END_REGION

REGION Network 73: PT-504 HIGH_SET VALIDATION TIME OVER_(SYSTEM STOP)
   RUNG wire#powerrail
      Contact( "TIMING_SECS_DB_13".DONE )
      { S7_Templates := "time_type := Time" } "IEC_Timer_0_DB_6".TOF(pt := T#1S, et =>)
      wire#w1
      Coil( "ALARM DB PLC 2"."PT-504 HIGH_SET VALIDATION TIME OVER_(SYSTEM STOP)" )
   END_RUNG
   RUNG wire#w1
      P_Trig( "P_TRIG".ARR[72] )
      S_Coil( "HOOTER" )
   END_RUNG
   // the same network as SCL:
   "IEC_Timer_0_DB_6".TOF(IN := "TIMING_SECS_DB_13".DONE, PT := T#1S);
   "ALARM DB PLC 2"."PT-504 HIGH_SET VALIDATION TIME OVER_(SYSTEM STOP)" := "IEC_Timer_0_DB_6".Q;
   #_w1 := "IEC_Timer_0_DB_6".Q AND NOT "P_TRIG".ARR[72];   // rising edge
   "P_TRIG".ARR[72] := "IEC_Timer_0_DB_6".Q;
   IF #_w1 THEN "HOOTER" := TRUE; END_IF;
END_REGION

REGION Network 74: EDI-501A CONCENTRATE OUT PRESSURE PT-505 HIGH
   RUNG wire#powerrail
      { S7_Templates := "SrcType := Int" } EQ_Contact(in1 := "INTERLOCK DB"."EDI PARAMETER BUFF"."PT-505 HIGH", in2 := 2)
      wire#w1
      Coil( "ALARM DB PLC 2"."EDI-501A CONCENTRATE OUT PRESSURE PT-505 HIGH" )
   END_RUNG
   RUNG wire#w1
      P_Trig( "P_TRIG".ARR[73] )
      S_Coil( "HOOTER" )
   END_RUNG
   // the same network as SCL:
   "ALARM DB PLC 2"."EDI-501A CONCENTRATE OUT PRESSURE PT-505 HIGH" := "INTERLOCK DB"."EDI PARAMETER BUFF"."PT-505 HIGH" = 2;
   #_w1 := "ALARM DB PLC 2"."EDI-501A CONCENTRATE OUT PRESSURE PT-505 HIGH" AND NOT "P_TRIG".ARR[73];   // rising edge
   "P_TRIG".ARR[73] := "ALARM DB PLC 2"."EDI-501A CONCENTRATE OUT PRESSURE PT-505 HIGH";
   IF #_w1 THEN "HOOTER" := TRUE; END_IF;
END_REGION

REGION Network 75: PT-505 HIGH_SET VALIDATION TIME OVER_(SYSTEM STOP)
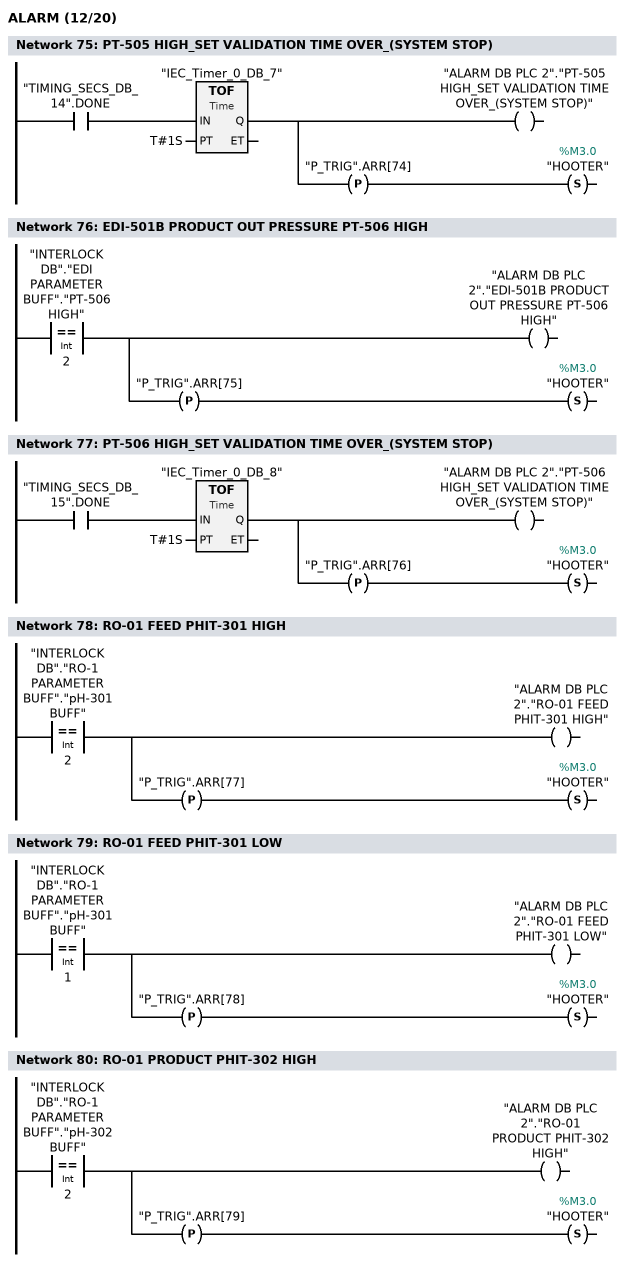
   RUNG wire#powerrail
      Contact( "TIMING_SECS_DB_14".DONE )
      { S7_Templates := "time_type := Time" } "IEC_Timer_0_DB_7".TOF(pt := T#1S, et =>)
      wire#w1
      Coil( "ALARM DB PLC 2"."PT-505 HIGH_SET VALIDATION TIME OVER_(SYSTEM STOP)" )
   END_RUNG
   RUNG wire#w1
      P_Trig( "P_TRIG".ARR[74] )
      S_Coil( "HOOTER" )
   END_RUNG
   // the same network as SCL:
   "IEC_Timer_0_DB_7".TOF(IN := "TIMING_SECS_DB_14".DONE, PT := T#1S);
   "ALARM DB PLC 2"."PT-505 HIGH_SET VALIDATION TIME OVER_(SYSTEM STOP)" := "IEC_Timer_0_DB_7".Q;
   #_w1 := "IEC_Timer_0_DB_7".Q AND NOT "P_TRIG".ARR[74];   // rising edge
   "P_TRIG".ARR[74] := "IEC_Timer_0_DB_7".Q;
   IF #_w1 THEN "HOOTER" := TRUE; END_IF;
END_REGION

REGION Network 76: EDI-501B PRODUCT OUT PRESSURE PT-506 HIGH
   RUNG wire#powerrail
      { S7_Templates := "SrcType := Int" } EQ_Contact(in1 := "INTERLOCK DB"."EDI PARAMETER BUFF"."PT-506 HIGH", in2 := 2)
      wire#w1
      Coil( "ALARM DB PLC 2"."EDI-501B PRODUCT OUT PRESSURE PT-506 HIGH" )
   END_RUNG
   RUNG wire#w1
      P_Trig( "P_TRIG".ARR[75] )
      S_Coil( "HOOTER" )
   END_RUNG
   // the same network as SCL:
   "ALARM DB PLC 2"."EDI-501B PRODUCT OUT PRESSURE PT-506 HIGH" := "INTERLOCK DB"."EDI PARAMETER BUFF"."PT-506 HIGH" = 2;
   #_w1 := "ALARM DB PLC 2"."EDI-501B PRODUCT OUT PRESSURE PT-506 HIGH" AND NOT "P_TRIG".ARR[75];   // rising edge
   "P_TRIG".ARR[75] := "ALARM DB PLC 2"."EDI-501B PRODUCT OUT PRESSURE PT-506 HIGH";
   IF #_w1 THEN "HOOTER" := TRUE; END_IF;
END_REGION

REGION Network 77: PT-506 HIGH_SET VALIDATION TIME OVER_(SYSTEM STOP)
   RUNG wire#powerrail
      Contact( "TIMING_SECS_DB_15".DONE )
      { S7_Templates := "time_type := Time" } "IEC_Timer_0_DB_8".TOF(pt := T#1S, et =>)
      wire#w1
      Coil( "ALARM DB PLC 2"."PT-506 HIGH_SET VALIDATION TIME OVER_(SYSTEM STOP)" )
   END_RUNG
   RUNG wire#w1
      P_Trig( "P_TRIG".ARR[76] )
      S_Coil( "HOOTER" )
   END_RUNG
   // the same network as SCL:
   "IEC_Timer_0_DB_8".TOF(IN := "TIMING_SECS_DB_15".DONE, PT := T#1S);
   "ALARM DB PLC 2"."PT-506 HIGH_SET VALIDATION TIME OVER_(SYSTEM STOP)" := "IEC_Timer_0_DB_8".Q;
   #_w1 := "IEC_Timer_0_DB_8".Q AND NOT "P_TRIG".ARR[76];   // rising edge
   "P_TRIG".ARR[76] := "IEC_Timer_0_DB_8".Q;
   IF #_w1 THEN "HOOTER" := TRUE; END_IF;
END_REGION

REGION Network 78: RO-01 FEED PHIT-301 HIGH
   RUNG wire#powerrail
      { S7_Templates := "SrcType := Int" } EQ_Contact(in1 := "INTERLOCK DB"."RO-1 PARAMETER BUFF"."pH-301 BUFF", in2 := 2)
      wire#w1
      Coil( "ALARM DB PLC 2"."RO-01 FEED PHIT-301 HIGH" )
   END_RUNG
   RUNG wire#w1
      P_Trig( "P_TRIG".ARR[77] )
      S_Coil( "HOOTER" )
   END_RUNG
   // the same network as SCL:
   "ALARM DB PLC 2"."RO-01 FEED PHIT-301 HIGH" := "INTERLOCK DB"."RO-1 PARAMETER BUFF"."pH-301 BUFF" = 2;
   #_w1 := "ALARM DB PLC 2"."RO-01 FEED PHIT-301 HIGH" AND NOT "P_TRIG".ARR[77];   // rising edge
   "P_TRIG".ARR[77] := "ALARM DB PLC 2"."RO-01 FEED PHIT-301 HIGH";
   IF #_w1 THEN "HOOTER" := TRUE; END_IF;
END_REGION

REGION Network 79: RO-01 FEED PHIT-301 LOW
   RUNG wire#powerrail
      { S7_Templates := "SrcType := Int" } EQ_Contact(in1 := "INTERLOCK DB"."RO-1 PARAMETER BUFF"."pH-301 BUFF", in2 := 1)
      wire#w1
      Coil( "ALARM DB PLC 2"."RO-01 FEED PHIT-301 LOW" )
   END_RUNG
   RUNG wire#w1
      P_Trig( "P_TRIG".ARR[78] )
      S_Coil( "HOOTER" )
   END_RUNG
   // the same network as SCL:
   "ALARM DB PLC 2"."RO-01 FEED PHIT-301 LOW" := "INTERLOCK DB"."RO-1 PARAMETER BUFF"."pH-301 BUFF" = 1;
   #_w1 := "ALARM DB PLC 2"."RO-01 FEED PHIT-301 LOW" AND NOT "P_TRIG".ARR[78];   // rising edge
   "P_TRIG".ARR[78] := "ALARM DB PLC 2"."RO-01 FEED PHIT-301 LOW";
   IF #_w1 THEN "HOOTER" := TRUE; END_IF;
END_REGION

REGION Network 80: RO-01 PRODUCT PHIT-302 HIGH
   RUNG wire#powerrail
      { S7_Templates := "SrcType := Int" } EQ_Contact(in1 := "INTERLOCK DB"."RO-1 PARAMETER BUFF"."pH-302 BUFF", in2 := 2)
      wire#w1
      Coil( "ALARM DB PLC 2"."RO-01 PRODUCT PHIT-302 HIGH" )
   END_RUNG
   RUNG wire#w1
      P_Trig( "P_TRIG".ARR[79] )
      S_Coil( "HOOTER" )
   END_RUNG
   // the same network as SCL:
   "ALARM DB PLC 2"."RO-01 PRODUCT PHIT-302 HIGH" := "INTERLOCK DB"."RO-1 PARAMETER BUFF"."pH-302 BUFF" = 2;
   #_w1 := "ALARM DB PLC 2"."RO-01 PRODUCT PHIT-302 HIGH" AND NOT "P_TRIG".ARR[79];   // rising edge
   "P_TRIG".ARR[79] := "ALARM DB PLC 2"."RO-01 PRODUCT PHIT-302 HIGH";
   IF #_w1 THEN "HOOTER" := TRUE; END_IF;
END_REGION

REGION Network 81: RO-01 PRODUCT PHIT-302 LOW
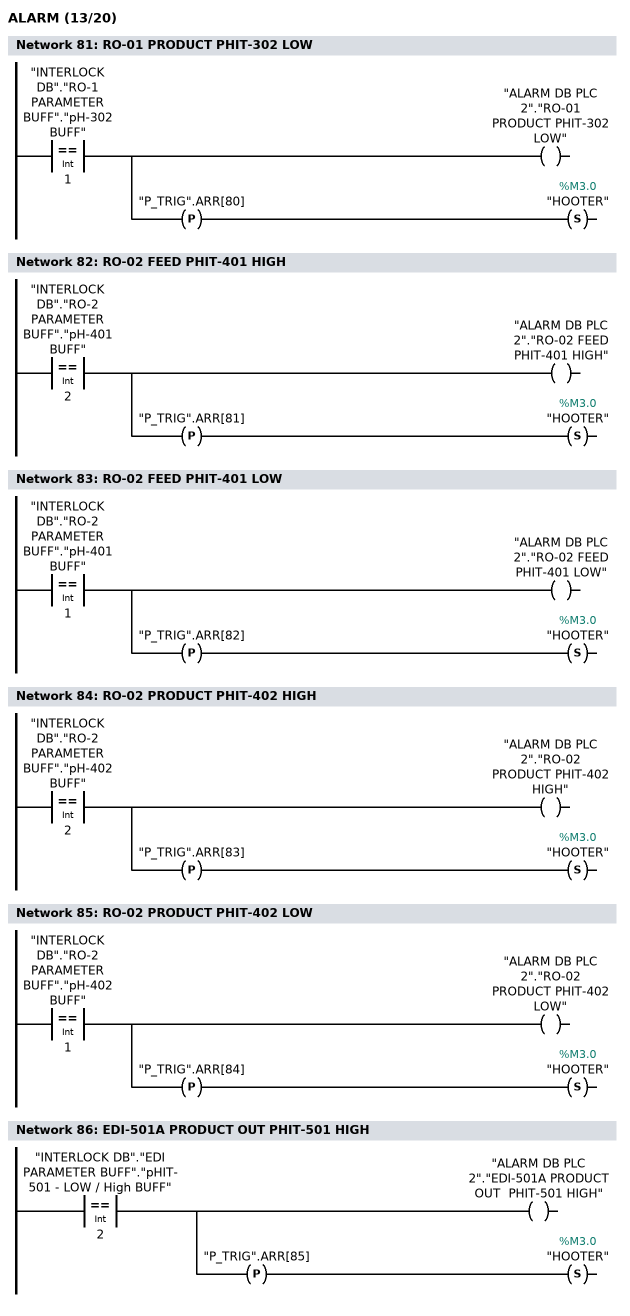
   RUNG wire#powerrail
      { S7_Templates := "SrcType := Int" } EQ_Contact(in1 := "INTERLOCK DB"."RO-1 PARAMETER BUFF"."pH-302 BUFF", in2 := 1)
      wire#w1
      Coil( "ALARM DB PLC 2"."RO-01 PRODUCT PHIT-302 LOW" )
   END_RUNG
   RUNG wire#w1
      P_Trig( "P_TRIG".ARR[80] )
      S_Coil( "HOOTER" )
   END_RUNG
   // the same network as SCL:
   "ALARM DB PLC 2"."RO-01 PRODUCT PHIT-302 LOW" := "INTERLOCK DB"."RO-1 PARAMETER BUFF"."pH-302 BUFF" = 1;
   #_w1 := "ALARM DB PLC 2"."RO-01 PRODUCT PHIT-302 LOW" AND NOT "P_TRIG".ARR[80];   // rising edge
   "P_TRIG".ARR[80] := "ALARM DB PLC 2"."RO-01 PRODUCT PHIT-302 LOW";
   IF #_w1 THEN "HOOTER" := TRUE; END_IF;
END_REGION

REGION Network 82: RO-02 FEED PHIT-401 HIGH
   RUNG wire#powerrail
      { S7_Templates := "SrcType := Int" } EQ_Contact(in1 := "INTERLOCK DB"."RO-2 PARAMETER BUFF"."pH-401 BUFF", in2 := 2)
      wire#w1
      Coil( "ALARM DB PLC 2"."RO-02 FEED PHIT-401 HIGH" )
   END_RUNG
   RUNG wire#w1
      P_Trig( "P_TRIG".ARR[81] )
      S_Coil( "HOOTER" )
   END_RUNG
   // the same network as SCL:
   "ALARM DB PLC 2"."RO-02 FEED PHIT-401 HIGH" := "INTERLOCK DB"."RO-2 PARAMETER BUFF"."pH-401 BUFF" = 2;
   #_w1 := "ALARM DB PLC 2"."RO-02 FEED PHIT-401 HIGH" AND NOT "P_TRIG".ARR[81];   // rising edge
   "P_TRIG".ARR[81] := "ALARM DB PLC 2"."RO-02 FEED PHIT-401 HIGH";
   IF #_w1 THEN "HOOTER" := TRUE; END_IF;
END_REGION

REGION Network 83: RO-02 FEED PHIT-401 LOW
   RUNG wire#powerrail
      { S7_Templates := "SrcType := Int" } EQ_Contact(in1 := "INTERLOCK DB"."RO-2 PARAMETER BUFF"."pH-401 BUFF", in2 := 1)
      wire#w1
      Coil( "ALARM DB PLC 2"."RO-02 FEED PHIT-401 LOW" )
   END_RUNG
   RUNG wire#w1
      P_Trig( "P_TRIG".ARR[82] )
      S_Coil( "HOOTER" )
   END_RUNG
   // the same network as SCL:
   "ALARM DB PLC 2"."RO-02 FEED PHIT-401 LOW" := "INTERLOCK DB"."RO-2 PARAMETER BUFF"."pH-401 BUFF" = 1;
   #_w1 := "ALARM DB PLC 2"."RO-02 FEED PHIT-401 LOW" AND NOT "P_TRIG".ARR[82];   // rising edge
   "P_TRIG".ARR[82] := "ALARM DB PLC 2"."RO-02 FEED PHIT-401 LOW";
   IF #_w1 THEN "HOOTER" := TRUE; END_IF;
END_REGION

REGION Network 84: RO-02 PRODUCT PHIT-402 HIGH
   RUNG wire#powerrail
      { S7_Templates := "SrcType := Int" } EQ_Contact(in1 := "INTERLOCK DB"."RO-2 PARAMETER BUFF"."pH-402 BUFF", in2 := 2)
      wire#w1
      Coil( "ALARM DB PLC 2"."RO-02 PRODUCT PHIT-402 HIGH" )
   END_RUNG
   RUNG wire#w1
      P_Trig( "P_TRIG".ARR[83] )
      S_Coil( "HOOTER" )
   END_RUNG
   // the same network as SCL:
   "ALARM DB PLC 2"."RO-02 PRODUCT PHIT-402 HIGH" := "INTERLOCK DB"."RO-2 PARAMETER BUFF"."pH-402 BUFF" = 2;
   #_w1 := "ALARM DB PLC 2"."RO-02 PRODUCT PHIT-402 HIGH" AND NOT "P_TRIG".ARR[83];   // rising edge
   "P_TRIG".ARR[83] := "ALARM DB PLC 2"."RO-02 PRODUCT PHIT-402 HIGH";
   IF #_w1 THEN "HOOTER" := TRUE; END_IF;
END_REGION

REGION Network 85: RO-02 PRODUCT PHIT-402 LOW
   RUNG wire#powerrail
      { S7_Templates := "SrcType := Int" } EQ_Contact(in1 := "INTERLOCK DB"."RO-2 PARAMETER BUFF"."pH-402 BUFF", in2 := 1)
      wire#w1
      Coil( "ALARM DB PLC 2"."RO-02 PRODUCT PHIT-402 LOW" )
   END_RUNG
   RUNG wire#w1
      P_Trig( "P_TRIG".ARR[84] )
      S_Coil( "HOOTER" )
   END_RUNG
   // the same network as SCL:
   "ALARM DB PLC 2"."RO-02 PRODUCT PHIT-402 LOW" := "INTERLOCK DB"."RO-2 PARAMETER BUFF"."pH-402 BUFF" = 1;
   #_w1 := "ALARM DB PLC 2"."RO-02 PRODUCT PHIT-402 LOW" AND NOT "P_TRIG".ARR[84];   // rising edge
   "P_TRIG".ARR[84] := "ALARM DB PLC 2"."RO-02 PRODUCT PHIT-402 LOW";
   IF #_w1 THEN "HOOTER" := TRUE; END_IF;
END_REGION

REGION Network 86: EDI-501A PRODUCT OUT PHIT-501 HIGH
   RUNG wire#powerrail
      { S7_Templates := "SrcType := Int" } EQ_Contact(in1 := "INTERLOCK DB"."EDI PARAMETER BUFF"."pHIT-501 - LOW / High BUFF", in2 := 2)
      wire#w1
      Coil( "ALARM DB PLC 2"."EDI-501A PRODUCT OUT  PHIT-501 HIGH" )
   END_RUNG
   RUNG wire#w1
      P_Trig( "P_TRIG".ARR[85] )
      S_Coil( "HOOTER" )
   END_RUNG
   // the same network as SCL:
   "ALARM DB PLC 2"."EDI-501A PRODUCT OUT  PHIT-501 HIGH" := "INTERLOCK DB"."EDI PARAMETER BUFF"."pHIT-501 - LOW / High BUFF" = 2;
   #_w1 := "ALARM DB PLC 2"."EDI-501A PRODUCT OUT  PHIT-501 HIGH" AND NOT "P_TRIG".ARR[85];   // rising edge
   "P_TRIG".ARR[85] := "ALARM DB PLC 2"."EDI-501A PRODUCT OUT  PHIT-501 HIGH";
   IF #_w1 THEN "HOOTER" := TRUE; END_IF;
END_REGION

REGION Network 87: EDI-501A PRODUCT OUT PHIT-501 LOW
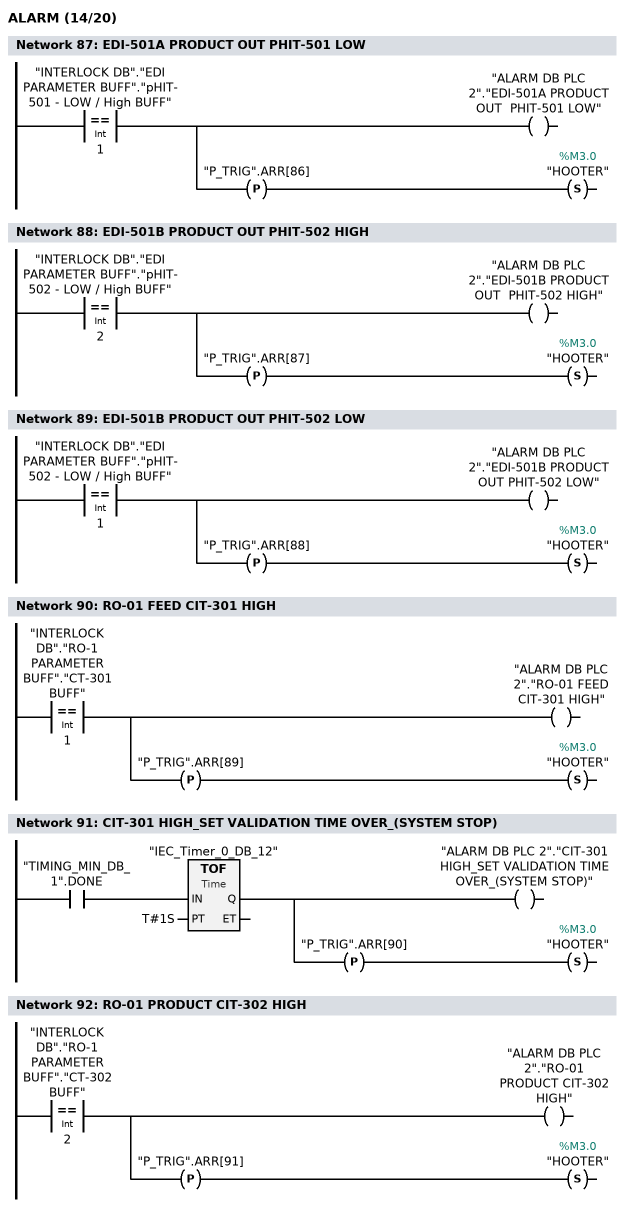
   RUNG wire#powerrail
      { S7_Templates := "SrcType := Int" } EQ_Contact(in1 := "INTERLOCK DB"."EDI PARAMETER BUFF"."pHIT-501 - LOW / High BUFF", in2 := 1)
      wire#w1
      Coil( "ALARM DB PLC 2"."EDI-501A PRODUCT OUT  PHIT-501 LOW" )
   END_RUNG
   RUNG wire#w1
      P_Trig( "P_TRIG".ARR[86] )
      S_Coil( "HOOTER" )
   END_RUNG
   // the same network as SCL:
   "ALARM DB PLC 2"."EDI-501A PRODUCT OUT  PHIT-501 LOW" := "INTERLOCK DB"."EDI PARAMETER BUFF"."pHIT-501 - LOW / High BUFF" = 1;
   #_w1 := "ALARM DB PLC 2"."EDI-501A PRODUCT OUT  PHIT-501 LOW" AND NOT "P_TRIG".ARR[86];   // rising edge
   "P_TRIG".ARR[86] := "ALARM DB PLC 2"."EDI-501A PRODUCT OUT  PHIT-501 LOW";
   IF #_w1 THEN "HOOTER" := TRUE; END_IF;
END_REGION

REGION Network 88: EDI-501B PRODUCT OUT PHIT-502 HIGH
   RUNG wire#powerrail
      { S7_Templates := "SrcType := Int" } EQ_Contact(in1 := "INTERLOCK DB"."EDI PARAMETER BUFF"."pHIT-502 - LOW / High BUFF", in2 := 2)
      wire#w1
      Coil( "ALARM DB PLC 2"."EDI-501B PRODUCT OUT  PHIT-502 HIGH" )
   END_RUNG
   RUNG wire#w1
      P_Trig( "P_TRIG".ARR[87] )
      S_Coil( "HOOTER" )
   END_RUNG
   // the same network as SCL:
   "ALARM DB PLC 2"."EDI-501B PRODUCT OUT  PHIT-502 HIGH" := "INTERLOCK DB"."EDI PARAMETER BUFF"."pHIT-502 - LOW / High BUFF" = 2;
   #_w1 := "ALARM DB PLC 2"."EDI-501B PRODUCT OUT  PHIT-502 HIGH" AND NOT "P_TRIG".ARR[87];   // rising edge
   "P_TRIG".ARR[87] := "ALARM DB PLC 2"."EDI-501B PRODUCT OUT  PHIT-502 HIGH";
   IF #_w1 THEN "HOOTER" := TRUE; END_IF;
END_REGION

REGION Network 89: EDI-501B PRODUCT OUT PHIT-502 LOW
   RUNG wire#powerrail
      { S7_Templates := "SrcType := Int" } EQ_Contact(in1 := "INTERLOCK DB"."EDI PARAMETER BUFF"."pHIT-502 - LOW / High BUFF", in2 := 1)
      wire#w1
      Coil( "ALARM DB PLC 2"."EDI-501B PRODUCT OUT PHIT-502 LOW" )
   END_RUNG
   RUNG wire#w1
      P_Trig( "P_TRIG".ARR[88] )
      S_Coil( "HOOTER" )
   END_RUNG
   // the same network as SCL:
   "ALARM DB PLC 2"."EDI-501B PRODUCT OUT PHIT-502 LOW" := "INTERLOCK DB"."EDI PARAMETER BUFF"."pHIT-502 - LOW / High BUFF" = 1;
   #_w1 := "ALARM DB PLC 2"."EDI-501B PRODUCT OUT PHIT-502 LOW" AND NOT "P_TRIG".ARR[88];   // rising edge
   "P_TRIG".ARR[88] := "ALARM DB PLC 2"."EDI-501B PRODUCT OUT PHIT-502 LOW";
   IF #_w1 THEN "HOOTER" := TRUE; END_IF;
END_REGION

REGION Network 90: RO-01 FEED CIT-301 HIGH
   RUNG wire#powerrail
      { S7_Templates := "SrcType := Int" } EQ_Contact(in1 := "INTERLOCK DB"."RO-1 PARAMETER BUFF"."CT-301 BUFF", in2 := 1)
      wire#w1
      Coil( "ALARM DB PLC 2"."RO-01 FEED CIT-301 HIGH" )
   END_RUNG
   RUNG wire#w1
      P_Trig( "P_TRIG".ARR[89] )
      S_Coil( "HOOTER" )
   END_RUNG
   // the same network as SCL:
   "ALARM DB PLC 2"."RO-01 FEED CIT-301 HIGH" := "INTERLOCK DB"."RO-1 PARAMETER BUFF"."CT-301 BUFF" = 1;
   #_w1 := "ALARM DB PLC 2"."RO-01 FEED CIT-301 HIGH" AND NOT "P_TRIG".ARR[89];   // rising edge
   "P_TRIG".ARR[89] := "ALARM DB PLC 2"."RO-01 FEED CIT-301 HIGH";
   IF #_w1 THEN "HOOTER" := TRUE; END_IF;
END_REGION

REGION Network 91: CIT-301 HIGH_SET VALIDATION TIME OVER_(SYSTEM STOP)
   RUNG wire#powerrail
      Contact( "TIMING_MIN_DB_1".DONE )
      { S7_Templates := "time_type := Time" } "IEC_Timer_0_DB_12".TOF(pt := T#1S, et =>)
      wire#w1
      Coil( "ALARM DB PLC 2"."CIT-301 HIGH_SET VALIDATION TIME OVER_(SYSTEM STOP)" )
   END_RUNG
   RUNG wire#w1
      P_Trig( "P_TRIG".ARR[90] )
      S_Coil( "HOOTER" )
   END_RUNG
   // the same network as SCL:
   "IEC_Timer_0_DB_12".TOF(IN := "TIMING_MIN_DB_1".DONE, PT := T#1S);
   "ALARM DB PLC 2"."CIT-301 HIGH_SET VALIDATION TIME OVER_(SYSTEM STOP)" := "IEC_Timer_0_DB_12".Q;
   #_w1 := "IEC_Timer_0_DB_12".Q AND NOT "P_TRIG".ARR[90];   // rising edge
   "P_TRIG".ARR[90] := "IEC_Timer_0_DB_12".Q;
   IF #_w1 THEN "HOOTER" := TRUE; END_IF;
END_REGION

REGION Network 92: RO-01 PRODUCT CIT-302 HIGH
   RUNG wire#powerrail
      { S7_Templates := "SrcType := Int" } EQ_Contact(in1 := "INTERLOCK DB"."RO-1 PARAMETER BUFF"."CT-302 BUFF", in2 := 2)
      wire#w1
      Coil( "ALARM DB PLC 2"."RO-01 PRODUCT CIT-302 HIGH" )
   END_RUNG
   RUNG wire#w1
      P_Trig( "P_TRIG".ARR[91] )
      S_Coil( "HOOTER" )
   END_RUNG
   // the same network as SCL:
   "ALARM DB PLC 2"."RO-01 PRODUCT CIT-302 HIGH" := "INTERLOCK DB"."RO-1 PARAMETER BUFF"."CT-302 BUFF" = 2;
   #_w1 := "ALARM DB PLC 2"."RO-01 PRODUCT CIT-302 HIGH" AND NOT "P_TRIG".ARR[91];   // rising edge
   "P_TRIG".ARR[91] := "ALARM DB PLC 2"."RO-01 PRODUCT CIT-302 HIGH";
   IF #_w1 THEN "HOOTER" := TRUE; END_IF;
END_REGION

REGION Network 93: CIT-302 HIGH_SET VALIDATION TIME OVER_(SYSTEM STOP)
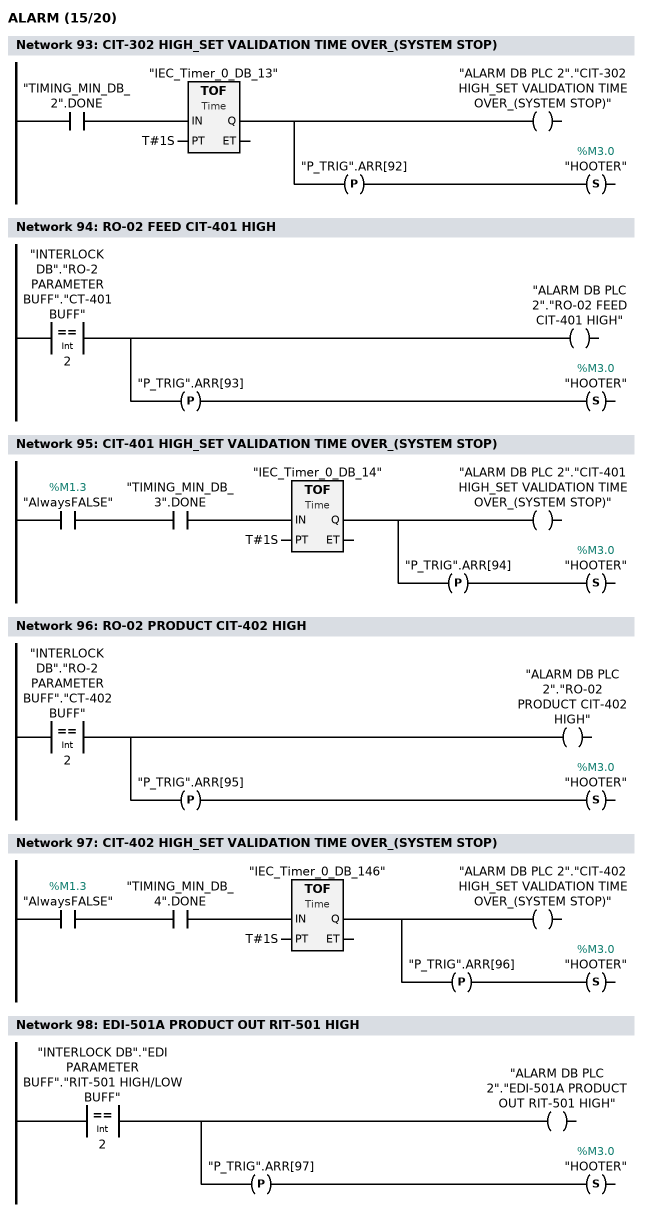
   RUNG wire#powerrail
      Contact( "TIMING_MIN_DB_2".DONE )
      { S7_Templates := "time_type := Time" } "IEC_Timer_0_DB_13".TOF(pt := T#1S, et =>)
      wire#w1
      Coil( "ALARM DB PLC 2"."CIT-302 HIGH_SET VALIDATION TIME OVER_(SYSTEM STOP)" )
   END_RUNG
   RUNG wire#w1
      P_Trig( "P_TRIG".ARR[92] )
      S_Coil( "HOOTER" )
   END_RUNG
   // the same network as SCL:
   "IEC_Timer_0_DB_13".TOF(IN := "TIMING_MIN_DB_2".DONE, PT := T#1S);
   "ALARM DB PLC 2"."CIT-302 HIGH_SET VALIDATION TIME OVER_(SYSTEM STOP)" := "IEC_Timer_0_DB_13".Q;
   #_w1 := "IEC_Timer_0_DB_13".Q AND NOT "P_TRIG".ARR[92];   // rising edge
   "P_TRIG".ARR[92] := "IEC_Timer_0_DB_13".Q;
   IF #_w1 THEN "HOOTER" := TRUE; END_IF;
END_REGION

REGION Network 94: RO-02 FEED CIT-401 HIGH
   RUNG wire#powerrail
      { S7_Templates := "SrcType := Int" } EQ_Contact(in1 := "INTERLOCK DB"."RO-2 PARAMETER BUFF"."CT-401 BUFF", in2 := 2)
      wire#w1
      Coil( "ALARM DB PLC 2"."RO-02 FEED CIT-401 HIGH" )
   END_RUNG
   RUNG wire#w1
      P_Trig( "P_TRIG".ARR[93] )
      S_Coil( "HOOTER" )
   END_RUNG
   // the same network as SCL:
   "ALARM DB PLC 2"."RO-02 FEED CIT-401 HIGH" := "INTERLOCK DB"."RO-2 PARAMETER BUFF"."CT-401 BUFF" = 2;
   #_w1 := "ALARM DB PLC 2"."RO-02 FEED CIT-401 HIGH" AND NOT "P_TRIG".ARR[93];   // rising edge
   "P_TRIG".ARR[93] := "ALARM DB PLC 2"."RO-02 FEED CIT-401 HIGH";
   IF #_w1 THEN "HOOTER" := TRUE; END_IF;
END_REGION

REGION Network 95: CIT-401 HIGH_SET VALIDATION TIME OVER_(SYSTEM STOP)
   RUNG wire#powerrail
      Contact( "AlwaysFALSE" )
      Contact( "TIMING_MIN_DB_3".DONE )
      { S7_Templates := "time_type := Time" } "IEC_Timer_0_DB_14".TOF(pt := T#1S, et =>)
      wire#w1
      Coil( "ALARM DB PLC 2"."CIT-401 HIGH_SET VALIDATION TIME OVER_(SYSTEM STOP)" )
   END_RUNG
   RUNG wire#w1
      P_Trig( "P_TRIG".ARR[94] )
      S_Coil( "HOOTER" )
   END_RUNG
   // the same network as SCL:
   "IEC_Timer_0_DB_14".TOF(IN := "AlwaysFALSE" AND "TIMING_MIN_DB_3".DONE, PT := T#1S);
   "ALARM DB PLC 2"."CIT-401 HIGH_SET VALIDATION TIME OVER_(SYSTEM STOP)" := "IEC_Timer_0_DB_14".Q;
   #_w1 := "IEC_Timer_0_DB_14".Q AND NOT "P_TRIG".ARR[94];   // rising edge
   "P_TRIG".ARR[94] := "IEC_Timer_0_DB_14".Q;
   IF #_w1 THEN "HOOTER" := TRUE; END_IF;
END_REGION

REGION Network 96: RO-02 PRODUCT CIT-402 HIGH
   RUNG wire#powerrail
      { S7_Templates := "SrcType := Int" } EQ_Contact(in1 := "INTERLOCK DB"."RO-2 PARAMETER BUFF"."CT-402 BUFF", in2 := 2)
      wire#w1
      Coil( "ALARM DB PLC 2"."RO-02 PRODUCT CIT-402 HIGH" )
   END_RUNG
   RUNG wire#w1
      P_Trig( "P_TRIG".ARR[95] )
      S_Coil( "HOOTER" )
   END_RUNG
   // the same network as SCL:
   "ALARM DB PLC 2"."RO-02 PRODUCT CIT-402 HIGH" := "INTERLOCK DB"."RO-2 PARAMETER BUFF"."CT-402 BUFF" = 2;
   #_w1 := "ALARM DB PLC 2"."RO-02 PRODUCT CIT-402 HIGH" AND NOT "P_TRIG".ARR[95];   // rising edge
   "P_TRIG".ARR[95] := "ALARM DB PLC 2"."RO-02 PRODUCT CIT-402 HIGH";
   IF #_w1 THEN "HOOTER" := TRUE; END_IF;
END_REGION

REGION Network 97: CIT-402 HIGH_SET VALIDATION TIME OVER_(SYSTEM STOP)
   RUNG wire#powerrail
      Contact( "AlwaysFALSE" )
      Contact( "TIMING_MIN_DB_4".DONE )
      { S7_Templates := "time_type := Time" } "IEC_Timer_0_DB_146".TOF(pt := T#1S, et =>)
      wire#w1
      Coil( "ALARM DB PLC 2"."CIT-402 HIGH_SET VALIDATION TIME OVER_(SYSTEM STOP)" )
   END_RUNG
   RUNG wire#w1
      P_Trig( "P_TRIG".ARR[96] )
      S_Coil( "HOOTER" )
   END_RUNG
   // the same network as SCL:
   "IEC_Timer_0_DB_146".TOF(IN := "AlwaysFALSE" AND "TIMING_MIN_DB_4".DONE, PT := T#1S);
   "ALARM DB PLC 2"."CIT-402 HIGH_SET VALIDATION TIME OVER_(SYSTEM STOP)" := "IEC_Timer_0_DB_146".Q;
   #_w1 := "IEC_Timer_0_DB_146".Q AND NOT "P_TRIG".ARR[96];   // rising edge
   "P_TRIG".ARR[96] := "IEC_Timer_0_DB_146".Q;
   IF #_w1 THEN "HOOTER" := TRUE; END_IF;
END_REGION

REGION Network 98: EDI-501A PRODUCT OUT RIT-501 HIGH
   RUNG wire#powerrail
      { S7_Templates := "SrcType := Int" } EQ_Contact(in1 := "INTERLOCK DB"."EDI PARAMETER BUFF"."RIT-501 HIGH/LOW BUFF", in2 := 2)
      wire#w1
      Coil( "ALARM DB PLC 2"."EDI-501A PRODUCT OUT RIT-501 HIGH" )
   END_RUNG
   RUNG wire#w1
      P_Trig( "P_TRIG".ARR[97] )
      S_Coil( "HOOTER" )
   END_RUNG
   // the same network as SCL:
   "ALARM DB PLC 2"."EDI-501A PRODUCT OUT RIT-501 HIGH" := "INTERLOCK DB"."EDI PARAMETER BUFF"."RIT-501 HIGH/LOW BUFF" = 2;
   #_w1 := "ALARM DB PLC 2"."EDI-501A PRODUCT OUT RIT-501 HIGH" AND NOT "P_TRIG".ARR[97];   // rising edge
   "P_TRIG".ARR[97] := "ALARM DB PLC 2"."EDI-501A PRODUCT OUT RIT-501 HIGH";
   IF #_w1 THEN "HOOTER" := TRUE; END_IF;
END_REGION

REGION Network 99: RIT-501A HIGH_SET VALIDATION TIME OVER_(SYSTEM STOP)
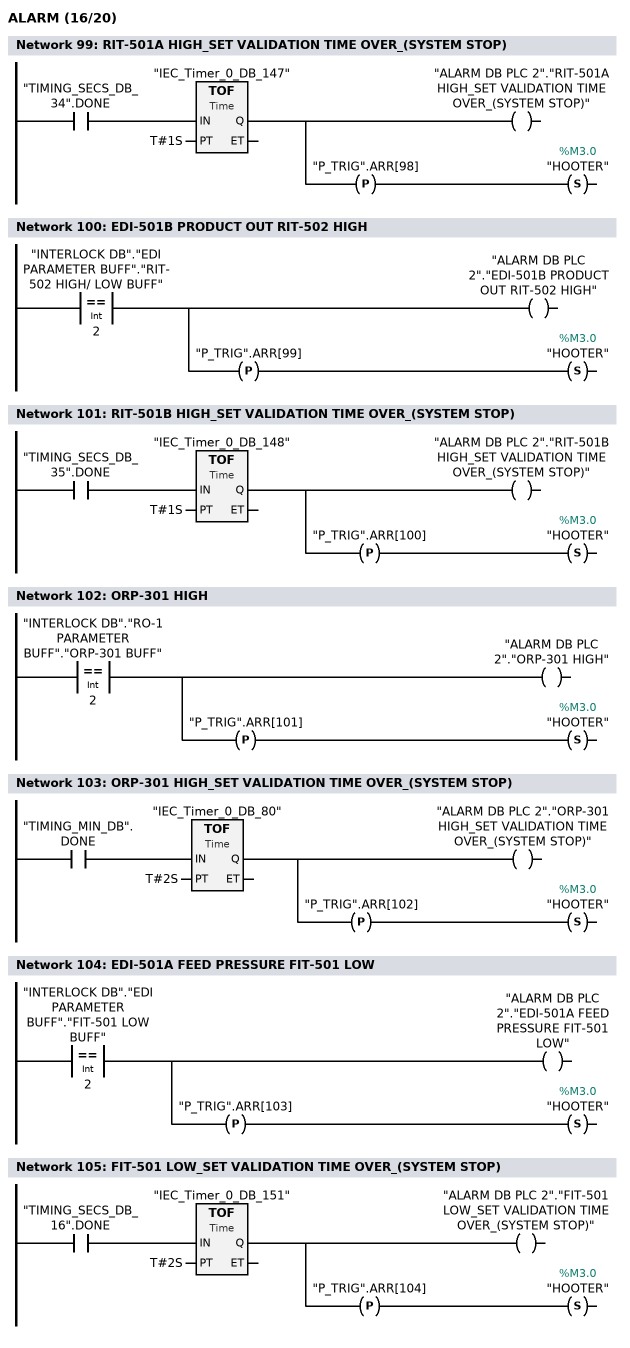
   RUNG wire#powerrail
      Contact( "TIMING_SECS_DB_34".DONE )
      { S7_Templates := "time_type := Time" } "IEC_Timer_0_DB_147".TOF(pt := T#1S, et =>)
      wire#w1
      Coil( "ALARM DB PLC 2"."RIT-501A HIGH_SET VALIDATION TIME OVER_(SYSTEM STOP)" )
   END_RUNG
   RUNG wire#w1
      P_Trig( "P_TRIG".ARR[98] )
      S_Coil( "HOOTER" )
   END_RUNG
   // the same network as SCL:
   "IEC_Timer_0_DB_147".TOF(IN := "TIMING_SECS_DB_34".DONE, PT := T#1S);
   "ALARM DB PLC 2"."RIT-501A HIGH_SET VALIDATION TIME OVER_(SYSTEM STOP)" := "IEC_Timer_0_DB_147".Q;
   #_w1 := "IEC_Timer_0_DB_147".Q AND NOT "P_TRIG".ARR[98];   // rising edge
   "P_TRIG".ARR[98] := "IEC_Timer_0_DB_147".Q;
   IF #_w1 THEN "HOOTER" := TRUE; END_IF;
END_REGION

REGION Network 100: EDI-501B PRODUCT OUT RIT-502 HIGH
   RUNG wire#powerrail
      { S7_Templates := "SrcType := Int" } EQ_Contact(in1 := "INTERLOCK DB"."EDI PARAMETER BUFF"."RIT-502 HIGH/ LOW BUFF", in2 := 2)
      wire#w1
      Coil( "ALARM DB PLC 2"."EDI-501B PRODUCT OUT RIT-502 HIGH" )
   END_RUNG
   RUNG wire#w1
      P_Trig( "P_TRIG".ARR[99] )
      S_Coil( "HOOTER" )
   END_RUNG
   // the same network as SCL:
   "ALARM DB PLC 2"."EDI-501B PRODUCT OUT RIT-502 HIGH" := "INTERLOCK DB"."EDI PARAMETER BUFF"."RIT-502 HIGH/ LOW BUFF" = 2;
   #_w1 := "ALARM DB PLC 2"."EDI-501B PRODUCT OUT RIT-502 HIGH" AND NOT "P_TRIG".ARR[99];   // rising edge
   "P_TRIG".ARR[99] := "ALARM DB PLC 2"."EDI-501B PRODUCT OUT RIT-502 HIGH";
   IF #_w1 THEN "HOOTER" := TRUE; END_IF;
END_REGION

REGION Network 101: RIT-501B HIGH_SET VALIDATION TIME OVER_(SYSTEM STOP)
   RUNG wire#powerrail
      Contact( "TIMING_SECS_DB_35".DONE )
      { S7_Templates := "time_type := Time" } "IEC_Timer_0_DB_148".TOF(pt := T#1S, et =>)
      wire#w1
      Coil( "ALARM DB PLC 2"."RIT-501B HIGH_SET VALIDATION TIME OVER_(SYSTEM STOP)" )
   END_RUNG
   RUNG wire#w1
      P_Trig( "P_TRIG".ARR[100] )
      S_Coil( "HOOTER" )
   END_RUNG
   // the same network as SCL:
   "IEC_Timer_0_DB_148".TOF(IN := "TIMING_SECS_DB_35".DONE, PT := T#1S);
   "ALARM DB PLC 2"."RIT-501B HIGH_SET VALIDATION TIME OVER_(SYSTEM STOP)" := "IEC_Timer_0_DB_148".Q;
   #_w1 := "IEC_Timer_0_DB_148".Q AND NOT "P_TRIG".ARR[100];   // rising edge
   "P_TRIG".ARR[100] := "IEC_Timer_0_DB_148".Q;
   IF #_w1 THEN "HOOTER" := TRUE; END_IF;
END_REGION

REGION Network 102: ORP-301 HIGH
   RUNG wire#powerrail
      { S7_Templates := "SrcType := Int" } EQ_Contact(in1 := "INTERLOCK DB"."RO-1 PARAMETER BUFF"."ORP-301 BUFF", in2 := 2)
      wire#w1
      Coil( "ALARM DB PLC 2"."ORP-301 HIGH" )
   END_RUNG
   RUNG wire#w1
      P_Trig( "P_TRIG".ARR[101] )
      S_Coil( "HOOTER" )
   END_RUNG
   // the same network as SCL:
   "ALARM DB PLC 2"."ORP-301 HIGH" := "INTERLOCK DB"."RO-1 PARAMETER BUFF"."ORP-301 BUFF" = 2;
   #_w1 := "ALARM DB PLC 2"."ORP-301 HIGH" AND NOT "P_TRIG".ARR[101];   // rising edge
   "P_TRIG".ARR[101] := "ALARM DB PLC 2"."ORP-301 HIGH";
   IF #_w1 THEN "HOOTER" := TRUE; END_IF;
END_REGION

REGION Network 103: ORP-301 HIGH_SET VALIDATION TIME OVER_(SYSTEM STOP)
   RUNG wire#powerrail
      Contact( "TIMING_MIN_DB".DONE )
      { S7_Templates := "time_type := Time" } "IEC_Timer_0_DB_80".TOF(pt := T#2S, et =>)
      wire#w1
      Coil( "ALARM DB PLC 2"."ORP-301 HIGH_SET VALIDATION TIME OVER_(SYSTEM STOP)" )
   END_RUNG
   RUNG wire#w1
      P_Trig( "P_TRIG".ARR[102] )
      S_Coil( "HOOTER" )
   END_RUNG
   // the same network as SCL:
   "IEC_Timer_0_DB_80".TOF(IN := "TIMING_MIN_DB".DONE, PT := T#2S);
   "ALARM DB PLC 2"."ORP-301 HIGH_SET VALIDATION TIME OVER_(SYSTEM STOP)" := "IEC_Timer_0_DB_80".Q;
   #_w1 := "IEC_Timer_0_DB_80".Q AND NOT "P_TRIG".ARR[102];   // rising edge
   "P_TRIG".ARR[102] := "IEC_Timer_0_DB_80".Q;
   IF #_w1 THEN "HOOTER" := TRUE; END_IF;
END_REGION

REGION Network 104: EDI-501A FEED PRESSURE FIT-501 LOW
   RUNG wire#powerrail
      { S7_Templates := "SrcType := Int" } EQ_Contact(in1 := "INTERLOCK DB"."EDI PARAMETER BUFF"."FIT-501 LOW BUFF", in2 := 2)
      wire#w1
      Coil( "ALARM DB PLC 2"."EDI-501A FEED PRESSURE FIT-501 LOW" )
   END_RUNG
   RUNG wire#w1
      P_Trig( "P_TRIG".ARR[103] )
      S_Coil( "HOOTER" )
   END_RUNG
   // the same network as SCL:
   "ALARM DB PLC 2"."EDI-501A FEED PRESSURE FIT-501 LOW" := "INTERLOCK DB"."EDI PARAMETER BUFF"."FIT-501 LOW BUFF" = 2;
   #_w1 := "ALARM DB PLC 2"."EDI-501A FEED PRESSURE FIT-501 LOW" AND NOT "P_TRIG".ARR[103];   // rising edge
   "P_TRIG".ARR[103] := "ALARM DB PLC 2"."EDI-501A FEED PRESSURE FIT-501 LOW";
   IF #_w1 THEN "HOOTER" := TRUE; END_IF;
END_REGION

REGION Network 105: FIT-501 LOW_SET VALIDATION TIME OVER_(SYSTEM STOP)
   RUNG wire#powerrail
      Contact( "TIMING_SECS_DB_16".DONE )
      { S7_Templates := "time_type := Time" } "IEC_Timer_0_DB_151".TOF(pt := T#2S, et =>)
      wire#w1
      Coil( "ALARM DB PLC 2"."FIT-501  LOW_SET VALIDATION TIME OVER_(SYSTEM STOP)" )
   END_RUNG
   RUNG wire#w1
      P_Trig( "P_TRIG".ARR[104] )
      S_Coil( "HOOTER" )
   END_RUNG
   // the same network as SCL:
   "IEC_Timer_0_DB_151".TOF(IN := "TIMING_SECS_DB_16".DONE, PT := T#2S);
   "ALARM DB PLC 2"."FIT-501  LOW_SET VALIDATION TIME OVER_(SYSTEM STOP)" := "IEC_Timer_0_DB_151".Q;
   #_w1 := "IEC_Timer_0_DB_151".Q AND NOT "P_TRIG".ARR[104];   // rising edge
   "P_TRIG".ARR[104] := "IEC_Timer_0_DB_151".Q;
   IF #_w1 THEN "HOOTER" := TRUE; END_IF;
END_REGION

REGION Network 106: EDI-501B FEED PRESSURE FIT-502 LOW
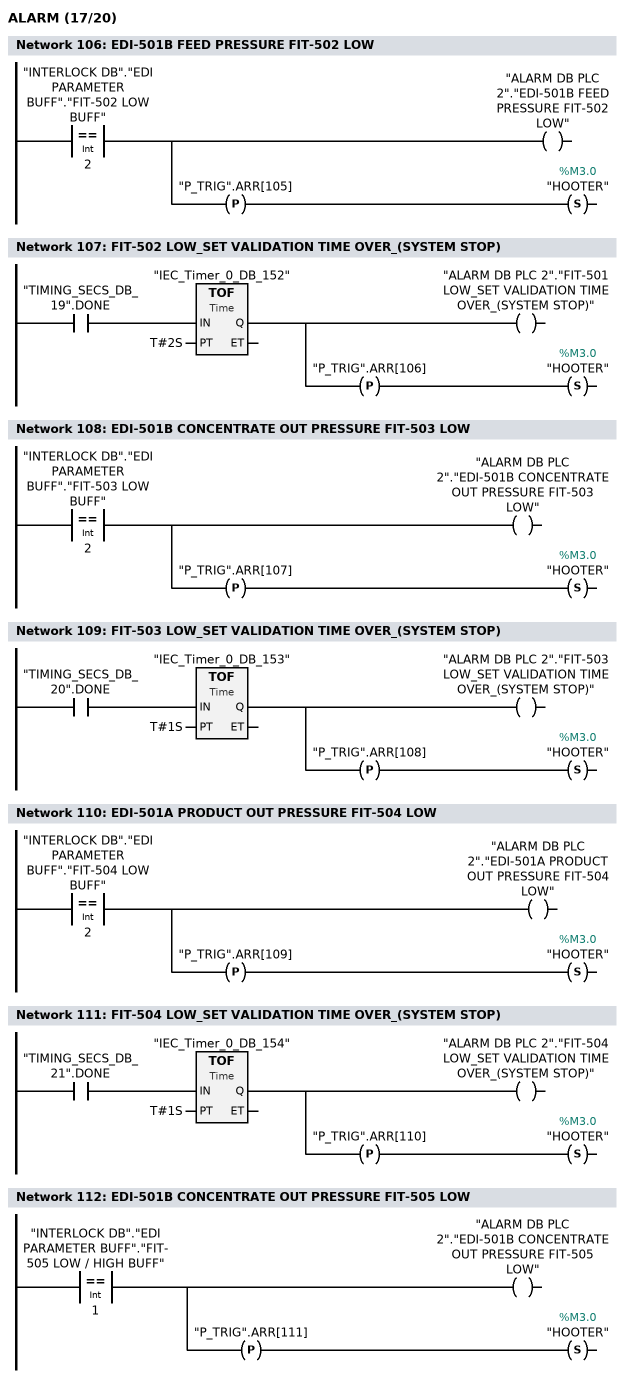
   RUNG wire#powerrail
      { S7_Templates := "SrcType := Int" } EQ_Contact(in1 := "INTERLOCK DB"."EDI PARAMETER BUFF"."FIT-502 LOW  BUFF", in2 := 2)
      wire#w1
      Coil( "ALARM DB PLC 2"."EDI-501B FEED PRESSURE FIT-502 LOW" )
   END_RUNG
   RUNG wire#w1
      P_Trig( "P_TRIG".ARR[105] )
      S_Coil( "HOOTER" )
   END_RUNG
   // the same network as SCL:
   "ALARM DB PLC 2"."EDI-501B FEED PRESSURE FIT-502 LOW" := "INTERLOCK DB"."EDI PARAMETER BUFF"."FIT-502 LOW  BUFF" = 2;
   #_w1 := "ALARM DB PLC 2"."EDI-501B FEED PRESSURE FIT-502 LOW" AND NOT "P_TRIG".ARR[105];   // rising edge
   "P_TRIG".ARR[105] := "ALARM DB PLC 2"."EDI-501B FEED PRESSURE FIT-502 LOW";
   IF #_w1 THEN "HOOTER" := TRUE; END_IF;
END_REGION

REGION Network 107: FIT-502 LOW_SET VALIDATION TIME OVER_(SYSTEM STOP)
   RUNG wire#powerrail
      Contact( "TIMING_SECS_DB_19".DONE )
      { S7_Templates := "time_type := Time" } "IEC_Timer_0_DB_152".TOF(pt := T#2S, et =>)
      wire#w1
      Coil( "ALARM DB PLC 2"."FIT-501 LOW_SET VALIDATION TIME OVER_(SYSTEM STOP)" )
   END_RUNG
   RUNG wire#w1
      P_Trig( "P_TRIG".ARR[106] )
      S_Coil( "HOOTER" )
   END_RUNG
   // the same network as SCL:
   "IEC_Timer_0_DB_152".TOF(IN := "TIMING_SECS_DB_19".DONE, PT := T#2S);
   "ALARM DB PLC 2"."FIT-501 LOW_SET VALIDATION TIME OVER_(SYSTEM STOP)" := "IEC_Timer_0_DB_152".Q;
   #_w1 := "IEC_Timer_0_DB_152".Q AND NOT "P_TRIG".ARR[106];   // rising edge
   "P_TRIG".ARR[106] := "IEC_Timer_0_DB_152".Q;
   IF #_w1 THEN "HOOTER" := TRUE; END_IF;
END_REGION

REGION Network 108: EDI-501B CONCENTRATE OUT PRESSURE FIT-503 LOW
   RUNG wire#powerrail
      { S7_Templates := "SrcType := Int" } EQ_Contact(in1 := "INTERLOCK DB"."EDI PARAMETER BUFF"."FIT-503 LOW BUFF", in2 := 2)
      wire#w1
      Coil( "ALARM DB PLC 2"."EDI-501B CONCENTRATE OUT PRESSURE FIT-503 LOW" )
   END_RUNG
   RUNG wire#w1
      P_Trig( "P_TRIG".ARR[107] )
      S_Coil( "HOOTER" )
   END_RUNG
   // the same network as SCL:
   "ALARM DB PLC 2"."EDI-501B CONCENTRATE OUT PRESSURE FIT-503 LOW" := "INTERLOCK DB"."EDI PARAMETER BUFF"."FIT-503 LOW BUFF" = 2;
   #_w1 := "ALARM DB PLC 2"."EDI-501B CONCENTRATE OUT PRESSURE FIT-503 LOW" AND NOT "P_TRIG".ARR[107];   // rising edge
   "P_TRIG".ARR[107] := "ALARM DB PLC 2"."EDI-501B CONCENTRATE OUT PRESSURE FIT-503 LOW";
   IF #_w1 THEN "HOOTER" := TRUE; END_IF;
END_REGION

REGION Network 109: FIT-503 LOW_SET VALIDATION TIME OVER_(SYSTEM STOP)
   RUNG wire#powerrail
      Contact( "TIMING_SECS_DB_20".DONE )
      { S7_Templates := "time_type := Time" } "IEC_Timer_0_DB_153".TOF(pt := T#1S, et =>)
      wire#w1
      Coil( "ALARM DB PLC 2"."FIT-503 LOW_SET VALIDATION TIME OVER_(SYSTEM STOP)" )
   END_RUNG
   RUNG wire#w1
      P_Trig( "P_TRIG".ARR[108] )
      S_Coil( "HOOTER" )
   END_RUNG
   // the same network as SCL:
   "IEC_Timer_0_DB_153".TOF(IN := "TIMING_SECS_DB_20".DONE, PT := T#1S);
   "ALARM DB PLC 2"."FIT-503 LOW_SET VALIDATION TIME OVER_(SYSTEM STOP)" := "IEC_Timer_0_DB_153".Q;
   #_w1 := "IEC_Timer_0_DB_153".Q AND NOT "P_TRIG".ARR[108];   // rising edge
   "P_TRIG".ARR[108] := "IEC_Timer_0_DB_153".Q;
   IF #_w1 THEN "HOOTER" := TRUE; END_IF;
END_REGION

REGION Network 110: EDI-501A PRODUCT OUT PRESSURE FIT-504 LOW
   RUNG wire#powerrail
      { S7_Templates := "SrcType := Int" } EQ_Contact(in1 := "INTERLOCK DB"."EDI PARAMETER BUFF"."FIT-504 LOW BUFF", in2 := 2)
      wire#w1
      Coil( "ALARM DB PLC 2"."EDI-501A PRODUCT OUT PRESSURE FIT-504 LOW" )
   END_RUNG
   RUNG wire#w1
      P_Trig( "P_TRIG".ARR[109] )
      S_Coil( "HOOTER" )
   END_RUNG
   // the same network as SCL:
   "ALARM DB PLC 2"."EDI-501A PRODUCT OUT PRESSURE FIT-504 LOW" := "INTERLOCK DB"."EDI PARAMETER BUFF"."FIT-504 LOW BUFF" = 2;
   #_w1 := "ALARM DB PLC 2"."EDI-501A PRODUCT OUT PRESSURE FIT-504 LOW" AND NOT "P_TRIG".ARR[109];   // rising edge
   "P_TRIG".ARR[109] := "ALARM DB PLC 2"."EDI-501A PRODUCT OUT PRESSURE FIT-504 LOW";
   IF #_w1 THEN "HOOTER" := TRUE; END_IF;
END_REGION

REGION Network 111: FIT-504 LOW_SET VALIDATION TIME OVER_(SYSTEM STOP)
   RUNG wire#powerrail
      Contact( "TIMING_SECS_DB_21".DONE )
      { S7_Templates := "time_type := Time" } "IEC_Timer_0_DB_154".TOF(pt := T#1S, et =>)
      wire#w1
      Coil( "ALARM DB PLC 2"."FIT-504 LOW_SET VALIDATION TIME OVER_(SYSTEM STOP)" )
   END_RUNG
   RUNG wire#w1
      P_Trig( "P_TRIG".ARR[110] )
      S_Coil( "HOOTER" )
   END_RUNG
   // the same network as SCL:
   "IEC_Timer_0_DB_154".TOF(IN := "TIMING_SECS_DB_21".DONE, PT := T#1S);
   "ALARM DB PLC 2"."FIT-504 LOW_SET VALIDATION TIME OVER_(SYSTEM STOP)" := "IEC_Timer_0_DB_154".Q;
   #_w1 := "IEC_Timer_0_DB_154".Q AND NOT "P_TRIG".ARR[110];   // rising edge
   "P_TRIG".ARR[110] := "IEC_Timer_0_DB_154".Q;
   IF #_w1 THEN "HOOTER" := TRUE; END_IF;
END_REGION

REGION Network 112: EDI-501B CONCENTRATE OUT PRESSURE FIT-505 LOW
   RUNG wire#powerrail
      { S7_Templates := "SrcType := Int" } EQ_Contact(in1 := "INTERLOCK DB"."EDI PARAMETER BUFF"."FIT-505 LOW / HIGH BUFF", in2 := 1)
      wire#w1
      Coil( "ALARM DB PLC 2"."EDI-501B CONCENTRATE OUT PRESSURE FIT-505 LOW" )
   END_RUNG
   RUNG wire#w1
      P_Trig( "P_TRIG".ARR[111] )
      S_Coil( "HOOTER" )
   END_RUNG
   // the same network as SCL:
   "ALARM DB PLC 2"."EDI-501B CONCENTRATE OUT PRESSURE FIT-505 LOW" := "INTERLOCK DB"."EDI PARAMETER BUFF"."FIT-505 LOW / HIGH BUFF" = 1;
   #_w1 := "ALARM DB PLC 2"."EDI-501B CONCENTRATE OUT PRESSURE FIT-505 LOW" AND NOT "P_TRIG".ARR[111];   // rising edge
   "P_TRIG".ARR[111] := "ALARM DB PLC 2"."EDI-501B CONCENTRATE OUT PRESSURE FIT-505 LOW";
   IF #_w1 THEN "HOOTER" := TRUE; END_IF;
END_REGION

REGION Network 113: FIT-505 LOW_SET VALIDATION TIME OVER_(SYSTEM STOP)
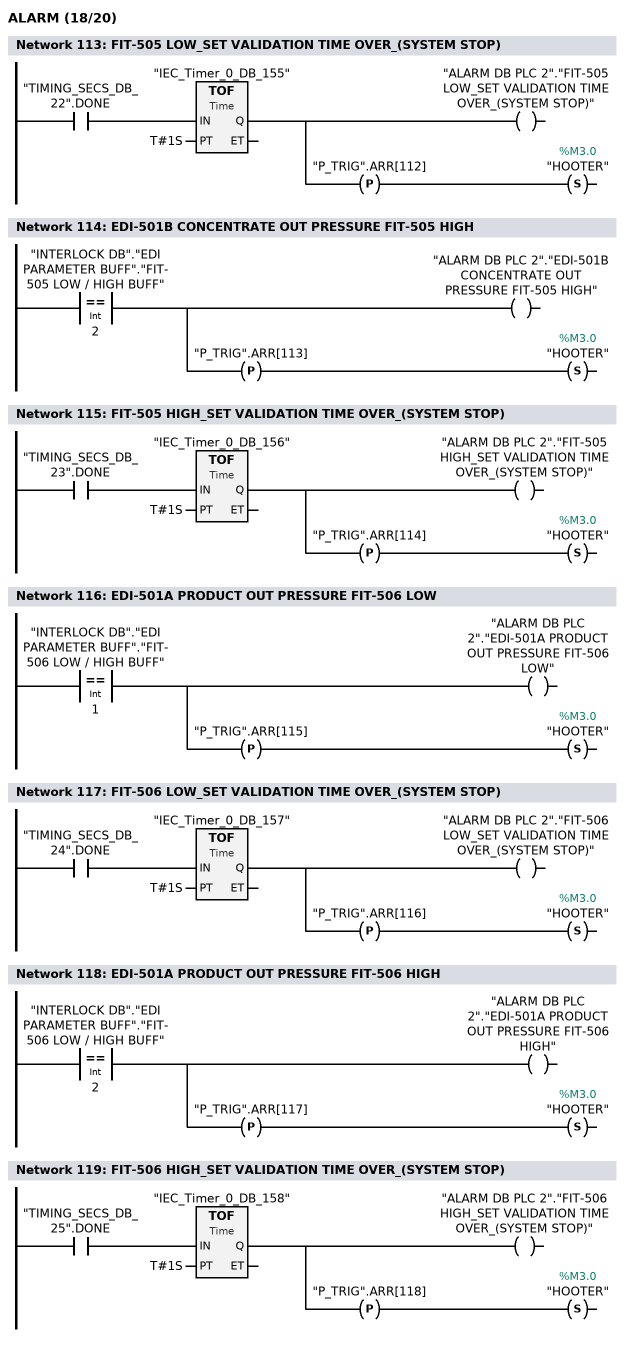
   RUNG wire#powerrail
      Contact( "TIMING_SECS_DB_22".DONE )
      { S7_Templates := "time_type := Time" } "IEC_Timer_0_DB_155".TOF(pt := T#1S, et =>)
      wire#w1
      Coil( "ALARM DB PLC 2"."FIT-505 LOW_SET VALIDATION TIME OVER_(SYSTEM STOP)" )
   END_RUNG
   RUNG wire#w1
      P_Trig( "P_TRIG".ARR[112] )
      S_Coil( "HOOTER" )
   END_RUNG
   // the same network as SCL:
   "IEC_Timer_0_DB_155".TOF(IN := "TIMING_SECS_DB_22".DONE, PT := T#1S);
   "ALARM DB PLC 2"."FIT-505 LOW_SET VALIDATION TIME OVER_(SYSTEM STOP)" := "IEC_Timer_0_DB_155".Q;
   #_w1 := "IEC_Timer_0_DB_155".Q AND NOT "P_TRIG".ARR[112];   // rising edge
   "P_TRIG".ARR[112] := "IEC_Timer_0_DB_155".Q;
   IF #_w1 THEN "HOOTER" := TRUE; END_IF;
END_REGION

REGION Network 114: EDI-501B CONCENTRATE OUT PRESSURE FIT-505 HIGH
   RUNG wire#powerrail
      { S7_Templates := "SrcType := Int" } EQ_Contact(in1 := "INTERLOCK DB"."EDI PARAMETER BUFF"."FIT-505 LOW / HIGH BUFF", in2 := 2)
      wire#w1
      Coil( "ALARM DB PLC 2"."EDI-501B CONCENTRATE OUT PRESSURE FIT-505 HIGH" )
   END_RUNG
   RUNG wire#w1
      P_Trig( "P_TRIG".ARR[113] )
      S_Coil( "HOOTER" )
   END_RUNG
   // the same network as SCL:
   "ALARM DB PLC 2"."EDI-501B CONCENTRATE OUT PRESSURE FIT-505 HIGH" := "INTERLOCK DB"."EDI PARAMETER BUFF"."FIT-505 LOW / HIGH BUFF" = 2;
   #_w1 := "ALARM DB PLC 2"."EDI-501B CONCENTRATE OUT PRESSURE FIT-505 HIGH" AND NOT "P_TRIG".ARR[113];   // rising edge
   "P_TRIG".ARR[113] := "ALARM DB PLC 2"."EDI-501B CONCENTRATE OUT PRESSURE FIT-505 HIGH";
   IF #_w1 THEN "HOOTER" := TRUE; END_IF;
END_REGION

REGION Network 115: FIT-505 HIGH_SET VALIDATION TIME OVER_(SYSTEM STOP)
   RUNG wire#powerrail
      Contact( "TIMING_SECS_DB_23".DONE )
      { S7_Templates := "time_type := Time" } "IEC_Timer_0_DB_156".TOF(pt := T#1S, et =>)
      wire#w1
      Coil( "ALARM DB PLC 2"."FIT-505 HIGH_SET VALIDATION TIME OVER_(SYSTEM STOP)" )
   END_RUNG
   RUNG wire#w1
      P_Trig( "P_TRIG".ARR[114] )
      S_Coil( "HOOTER" )
   END_RUNG
   // the same network as SCL:
   "IEC_Timer_0_DB_156".TOF(IN := "TIMING_SECS_DB_23".DONE, PT := T#1S);
   "ALARM DB PLC 2"."FIT-505 HIGH_SET VALIDATION TIME OVER_(SYSTEM STOP)" := "IEC_Timer_0_DB_156".Q;
   #_w1 := "IEC_Timer_0_DB_156".Q AND NOT "P_TRIG".ARR[114];   // rising edge
   "P_TRIG".ARR[114] := "IEC_Timer_0_DB_156".Q;
   IF #_w1 THEN "HOOTER" := TRUE; END_IF;
END_REGION

REGION Network 116: EDI-501A PRODUCT OUT PRESSURE FIT-506 LOW
   RUNG wire#powerrail
      { S7_Templates := "SrcType := Int" } EQ_Contact(in1 := "INTERLOCK DB"."EDI PARAMETER BUFF"."FIT-506 LOW / HIGH BUFF", in2 := 1)
      wire#w1
      Coil( "ALARM DB PLC 2"."EDI-501A PRODUCT OUT PRESSURE FIT-506 LOW" )
   END_RUNG
   RUNG wire#w1
      P_Trig( "P_TRIG".ARR[115] )
      S_Coil( "HOOTER" )
   END_RUNG
   // the same network as SCL:
   "ALARM DB PLC 2"."EDI-501A PRODUCT OUT PRESSURE FIT-506 LOW" := "INTERLOCK DB"."EDI PARAMETER BUFF"."FIT-506 LOW / HIGH BUFF" = 1;
   #_w1 := "ALARM DB PLC 2"."EDI-501A PRODUCT OUT PRESSURE FIT-506 LOW" AND NOT "P_TRIG".ARR[115];   // rising edge
   "P_TRIG".ARR[115] := "ALARM DB PLC 2"."EDI-501A PRODUCT OUT PRESSURE FIT-506 LOW";
   IF #_w1 THEN "HOOTER" := TRUE; END_IF;
END_REGION

REGION Network 117: FIT-506 LOW_SET VALIDATION TIME OVER_(SYSTEM STOP)
   RUNG wire#powerrail
      Contact( "TIMING_SECS_DB_24".DONE )
      { S7_Templates := "time_type := Time" } "IEC_Timer_0_DB_157".TOF(pt := T#1S, et =>)
      wire#w1
      Coil( "ALARM DB PLC 2"."FIT-506 LOW_SET VALIDATION TIME OVER_(SYSTEM STOP)" )
   END_RUNG
   RUNG wire#w1
      P_Trig( "P_TRIG".ARR[116] )
      S_Coil( "HOOTER" )
   END_RUNG
   // the same network as SCL:
   "IEC_Timer_0_DB_157".TOF(IN := "TIMING_SECS_DB_24".DONE, PT := T#1S);
   "ALARM DB PLC 2"."FIT-506 LOW_SET VALIDATION TIME OVER_(SYSTEM STOP)" := "IEC_Timer_0_DB_157".Q;
   #_w1 := "IEC_Timer_0_DB_157".Q AND NOT "P_TRIG".ARR[116];   // rising edge
   "P_TRIG".ARR[116] := "IEC_Timer_0_DB_157".Q;
   IF #_w1 THEN "HOOTER" := TRUE; END_IF;
END_REGION

REGION Network 118: EDI-501A PRODUCT OUT PRESSURE FIT-506 HIGH
   RUNG wire#powerrail
      { S7_Templates := "SrcType := Int" } EQ_Contact(in1 := "INTERLOCK DB"."EDI PARAMETER BUFF"."FIT-506 LOW / HIGH BUFF", in2 := 2)
      wire#w1
      Coil( "ALARM DB PLC 2"."EDI-501A PRODUCT OUT PRESSURE FIT-506 HIGH" )
   END_RUNG
   RUNG wire#w1
      P_Trig( "P_TRIG".ARR[117] )
      S_Coil( "HOOTER" )
   END_RUNG
   // the same network as SCL:
   "ALARM DB PLC 2"."EDI-501A PRODUCT OUT PRESSURE FIT-506 HIGH" := "INTERLOCK DB"."EDI PARAMETER BUFF"."FIT-506 LOW / HIGH BUFF" = 2;
   #_w1 := "ALARM DB PLC 2"."EDI-501A PRODUCT OUT PRESSURE FIT-506 HIGH" AND NOT "P_TRIG".ARR[117];   // rising edge
   "P_TRIG".ARR[117] := "ALARM DB PLC 2"."EDI-501A PRODUCT OUT PRESSURE FIT-506 HIGH";
   IF #_w1 THEN "HOOTER" := TRUE; END_IF;
END_REGION

REGION Network 119: FIT-506 HIGH_SET VALIDATION TIME OVER_(SYSTEM STOP)
   RUNG wire#powerrail
      Contact( "TIMING_SECS_DB_25".DONE )
      { S7_Templates := "time_type := Time" } "IEC_Timer_0_DB_158".TOF(pt := T#1S, et =>)
      wire#w1
      Coil( "ALARM DB PLC 2"."FIT-506 HIGH_SET VALIDATION TIME OVER_(SYSTEM STOP)" )
   END_RUNG
   RUNG wire#w1
      P_Trig( "P_TRIG".ARR[118] )
      S_Coil( "HOOTER" )
   END_RUNG
   // the same network as SCL:
   "IEC_Timer_0_DB_158".TOF(IN := "TIMING_SECS_DB_25".DONE, PT := T#1S);
   "ALARM DB PLC 2"."FIT-506 HIGH_SET VALIDATION TIME OVER_(SYSTEM STOP)" := "IEC_Timer_0_DB_158".Q;
   #_w1 := "IEC_Timer_0_DB_158".Q AND NOT "P_TRIG".ARR[118];   // rising edge
   "P_TRIG".ARR[118] := "IEC_Timer_0_DB_158".Q;
   IF #_w1 THEN "HOOTER" := TRUE; END_IF;
END_REGION

REGION Network 120: EDI-501B CONCENTRATE OUT PRESSURE FIT-507 LOW
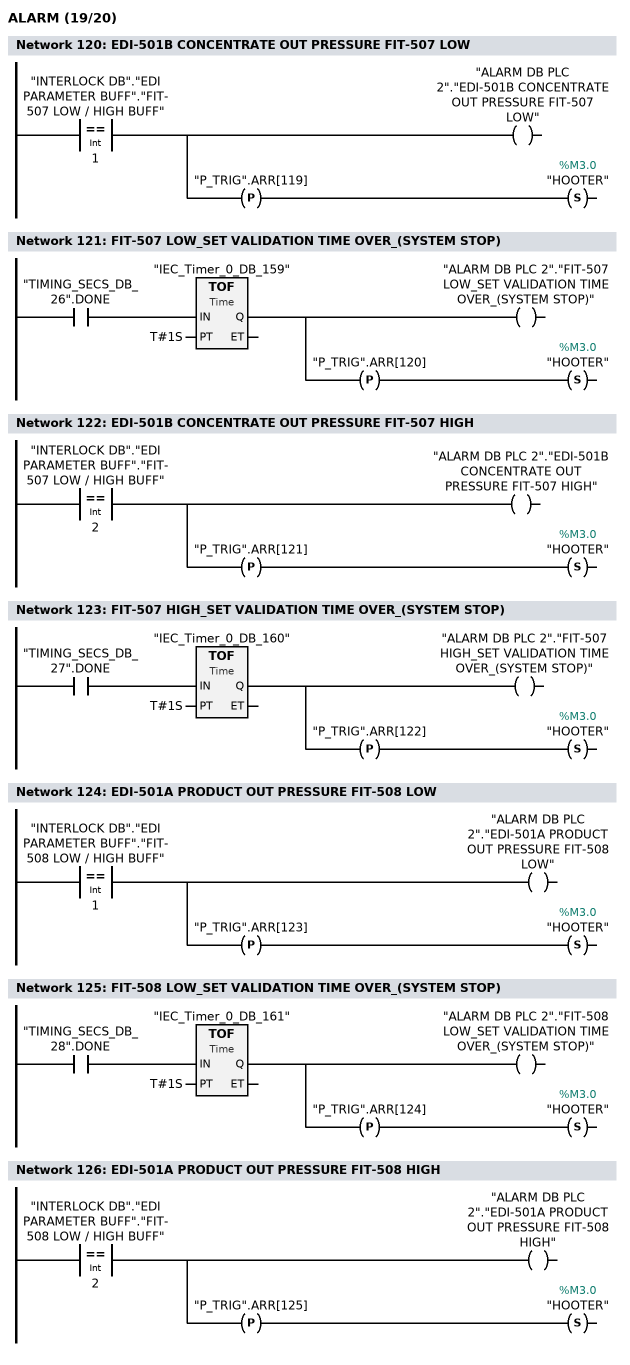
   RUNG wire#powerrail
      { S7_Templates := "SrcType := Int" } EQ_Contact(in1 := "INTERLOCK DB"."EDI PARAMETER BUFF"."FIT-507 LOW / HIGH BUFF", in2 := 1)
      wire#w1
      Coil( "ALARM DB PLC 2"."EDI-501B CONCENTRATE OUT PRESSURE FIT-507 LOW" )
   END_RUNG
   RUNG wire#w1
      P_Trig( "P_TRIG".ARR[119] )
      S_Coil( "HOOTER" )
   END_RUNG
   // the same network as SCL:
   "ALARM DB PLC 2"."EDI-501B CONCENTRATE OUT PRESSURE FIT-507 LOW" := "INTERLOCK DB"."EDI PARAMETER BUFF"."FIT-507 LOW / HIGH BUFF" = 1;
   #_w1 := "ALARM DB PLC 2"."EDI-501B CONCENTRATE OUT PRESSURE FIT-507 LOW" AND NOT "P_TRIG".ARR[119];   // rising edge
   "P_TRIG".ARR[119] := "ALARM DB PLC 2"."EDI-501B CONCENTRATE OUT PRESSURE FIT-507 LOW";
   IF #_w1 THEN "HOOTER" := TRUE; END_IF;
END_REGION

REGION Network 121: FIT-507 LOW_SET VALIDATION TIME OVER_(SYSTEM STOP)
   RUNG wire#powerrail
      Contact( "TIMING_SECS_DB_26".DONE )
      { S7_Templates := "time_type := Time" } "IEC_Timer_0_DB_159".TOF(pt := T#1S, et =>)
      wire#w1
      Coil( "ALARM DB PLC 2"."FIT-507 LOW_SET VALIDATION TIME OVER_(SYSTEM STOP)" )
   END_RUNG
   RUNG wire#w1
      P_Trig( "P_TRIG".ARR[120] )
      S_Coil( "HOOTER" )
   END_RUNG
   // the same network as SCL:
   "IEC_Timer_0_DB_159".TOF(IN := "TIMING_SECS_DB_26".DONE, PT := T#1S);
   "ALARM DB PLC 2"."FIT-507 LOW_SET VALIDATION TIME OVER_(SYSTEM STOP)" := "IEC_Timer_0_DB_159".Q;
   #_w1 := "IEC_Timer_0_DB_159".Q AND NOT "P_TRIG".ARR[120];   // rising edge
   "P_TRIG".ARR[120] := "IEC_Timer_0_DB_159".Q;
   IF #_w1 THEN "HOOTER" := TRUE; END_IF;
END_REGION

REGION Network 122: EDI-501B CONCENTRATE OUT PRESSURE FIT-507 HIGH
   RUNG wire#powerrail
      { S7_Templates := "SrcType := Int" } EQ_Contact(in1 := "INTERLOCK DB"."EDI PARAMETER BUFF"."FIT-507 LOW / HIGH BUFF", in2 := 2)
      wire#w1
      Coil( "ALARM DB PLC 2"."EDI-501B CONCENTRATE OUT PRESSURE FIT-507 HIGH" )
   END_RUNG
   RUNG wire#w1
      P_Trig( "P_TRIG".ARR[121] )
      S_Coil( "HOOTER" )
   END_RUNG
   // the same network as SCL:
   "ALARM DB PLC 2"."EDI-501B CONCENTRATE OUT PRESSURE FIT-507 HIGH" := "INTERLOCK DB"."EDI PARAMETER BUFF"."FIT-507 LOW / HIGH BUFF" = 2;
   #_w1 := "ALARM DB PLC 2"."EDI-501B CONCENTRATE OUT PRESSURE FIT-507 HIGH" AND NOT "P_TRIG".ARR[121];   // rising edge
   "P_TRIG".ARR[121] := "ALARM DB PLC 2"."EDI-501B CONCENTRATE OUT PRESSURE FIT-507 HIGH";
   IF #_w1 THEN "HOOTER" := TRUE; END_IF;
END_REGION

REGION Network 123: FIT-507 HIGH_SET VALIDATION TIME OVER_(SYSTEM STOP)
   RUNG wire#powerrail
      Contact( "TIMING_SECS_DB_27".DONE )
      { S7_Templates := "time_type := Time" } "IEC_Timer_0_DB_160".TOF(pt := T#1S, et =>)
      wire#w1
      Coil( "ALARM DB PLC 2"."FIT-507 HIGH_SET VALIDATION TIME OVER_(SYSTEM STOP)" )
   END_RUNG
   RUNG wire#w1
      P_Trig( "P_TRIG".ARR[122] )
      S_Coil( "HOOTER" )
   END_RUNG
   // the same network as SCL:
   "IEC_Timer_0_DB_160".TOF(IN := "TIMING_SECS_DB_27".DONE, PT := T#1S);
   "ALARM DB PLC 2"."FIT-507 HIGH_SET VALIDATION TIME OVER_(SYSTEM STOP)" := "IEC_Timer_0_DB_160".Q;
   #_w1 := "IEC_Timer_0_DB_160".Q AND NOT "P_TRIG".ARR[122];   // rising edge
   "P_TRIG".ARR[122] := "IEC_Timer_0_DB_160".Q;
   IF #_w1 THEN "HOOTER" := TRUE; END_IF;
END_REGION

REGION Network 124: EDI-501A PRODUCT OUT PRESSURE FIT-508 LOW
   RUNG wire#powerrail
      { S7_Templates := "SrcType := Int" } EQ_Contact(in1 := "INTERLOCK DB"."EDI PARAMETER BUFF"."FIT-508 LOW / HIGH BUFF", in2 := 1)
      wire#w1
      Coil( "ALARM DB PLC 2"."EDI-501A PRODUCT OUT PRESSURE FIT-508 LOW" )
   END_RUNG
   RUNG wire#w1
      P_Trig( "P_TRIG".ARR[123] )
      S_Coil( "HOOTER" )
   END_RUNG
   // the same network as SCL:
   "ALARM DB PLC 2"."EDI-501A PRODUCT OUT PRESSURE FIT-508 LOW" := "INTERLOCK DB"."EDI PARAMETER BUFF"."FIT-508 LOW / HIGH BUFF" = 1;
   #_w1 := "ALARM DB PLC 2"."EDI-501A PRODUCT OUT PRESSURE FIT-508 LOW" AND NOT "P_TRIG".ARR[123];   // rising edge
   "P_TRIG".ARR[123] := "ALARM DB PLC 2"."EDI-501A PRODUCT OUT PRESSURE FIT-508 LOW";
   IF #_w1 THEN "HOOTER" := TRUE; END_IF;
END_REGION

REGION Network 125: FIT-508 LOW_SET VALIDATION TIME OVER_(SYSTEM STOP)
   RUNG wire#powerrail
      Contact( "TIMING_SECS_DB_28".DONE )
      { S7_Templates := "time_type := Time" } "IEC_Timer_0_DB_161".TOF(pt := T#1S, et =>)
      wire#w1
      Coil( "ALARM DB PLC 2"."FIT-508 LOW_SET VALIDATION TIME OVER_(SYSTEM STOP)" )
   END_RUNG
   RUNG wire#w1
      P_Trig( "P_TRIG".ARR[124] )
      S_Coil( "HOOTER" )
   END_RUNG
   // the same network as SCL:
   "IEC_Timer_0_DB_161".TOF(IN := "TIMING_SECS_DB_28".DONE, PT := T#1S);
   "ALARM DB PLC 2"."FIT-508 LOW_SET VALIDATION TIME OVER_(SYSTEM STOP)" := "IEC_Timer_0_DB_161".Q;
   #_w1 := "IEC_Timer_0_DB_161".Q AND NOT "P_TRIG".ARR[124];   // rising edge
   "P_TRIG".ARR[124] := "IEC_Timer_0_DB_161".Q;
   IF #_w1 THEN "HOOTER" := TRUE; END_IF;
END_REGION

REGION Network 126: EDI-501A PRODUCT OUT PRESSURE FIT-508 HIGH
   RUNG wire#powerrail
      { S7_Templates := "SrcType := Int" } EQ_Contact(in1 := "INTERLOCK DB"."EDI PARAMETER BUFF"."FIT-508 LOW / HIGH BUFF", in2 := 2)
      wire#w1
      Coil( "ALARM DB PLC 2"."EDI-501A PRODUCT OUT PRESSURE FIT-508 HIGH" )
   END_RUNG
   RUNG wire#w1
      P_Trig( "P_TRIG".ARR[125] )
      S_Coil( "HOOTER" )
   END_RUNG
   // the same network as SCL:
   "ALARM DB PLC 2"."EDI-501A PRODUCT OUT PRESSURE FIT-508 HIGH" := "INTERLOCK DB"."EDI PARAMETER BUFF"."FIT-508 LOW / HIGH BUFF" = 2;
   #_w1 := "ALARM DB PLC 2"."EDI-501A PRODUCT OUT PRESSURE FIT-508 HIGH" AND NOT "P_TRIG".ARR[125];   // rising edge
   "P_TRIG".ARR[125] := "ALARM DB PLC 2"."EDI-501A PRODUCT OUT PRESSURE FIT-508 HIGH";
   IF #_w1 THEN "HOOTER" := TRUE; END_IF;
END_REGION

REGION Network 127: FIT-508 HIGH_SET VALIDATION TIME OVER_(SYSTEM STOP)
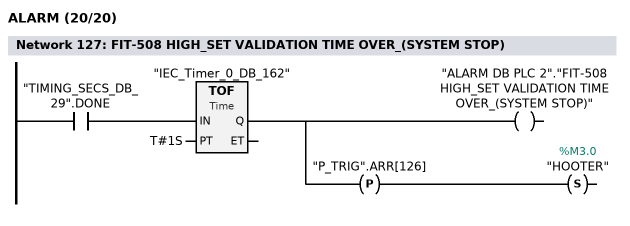
   RUNG wire#powerrail
      Contact( "TIMING_SECS_DB_29".DONE )
      { S7_Templates := "time_type := Time" } "IEC_Timer_0_DB_162".TOF(pt := T#1S, et =>)
      wire#w1
      Coil( "ALARM DB PLC 2"."FIT-508 HIGH_SET VALIDATION TIME OVER_(SYSTEM STOP)" )
   END_RUNG
   RUNG wire#w1
      P_Trig( "P_TRIG".ARR[126] )
      S_Coil( "HOOTER" )
   END_RUNG
   // the same network as SCL:
   "IEC_Timer_0_DB_162".TOF(IN := "TIMING_SECS_DB_29".DONE, PT := T#1S);
   "ALARM DB PLC 2"."FIT-508 HIGH_SET VALIDATION TIME OVER_(SYSTEM STOP)" := "IEC_Timer_0_DB_162".Q;
   #_w1 := "IEC_Timer_0_DB_162".Q AND NOT "P_TRIG".ARR[126];   // rising edge
   "P_TRIG".ARR[126] := "IEC_Timer_0_DB_162".Q;
   IF #_w1 THEN "HOOTER" := TRUE; END_IF;
END_REGION
END_FUNCTION

FUNCTION "AI SCALING" : Void   // FC5, LAD
{ S7_Optimized_Access := 'TRUE' }
// stored: SetENOAutomatically false
BEGIN

REGION Network 1: OXIDATION REDUCTION POTENTIO METER 301
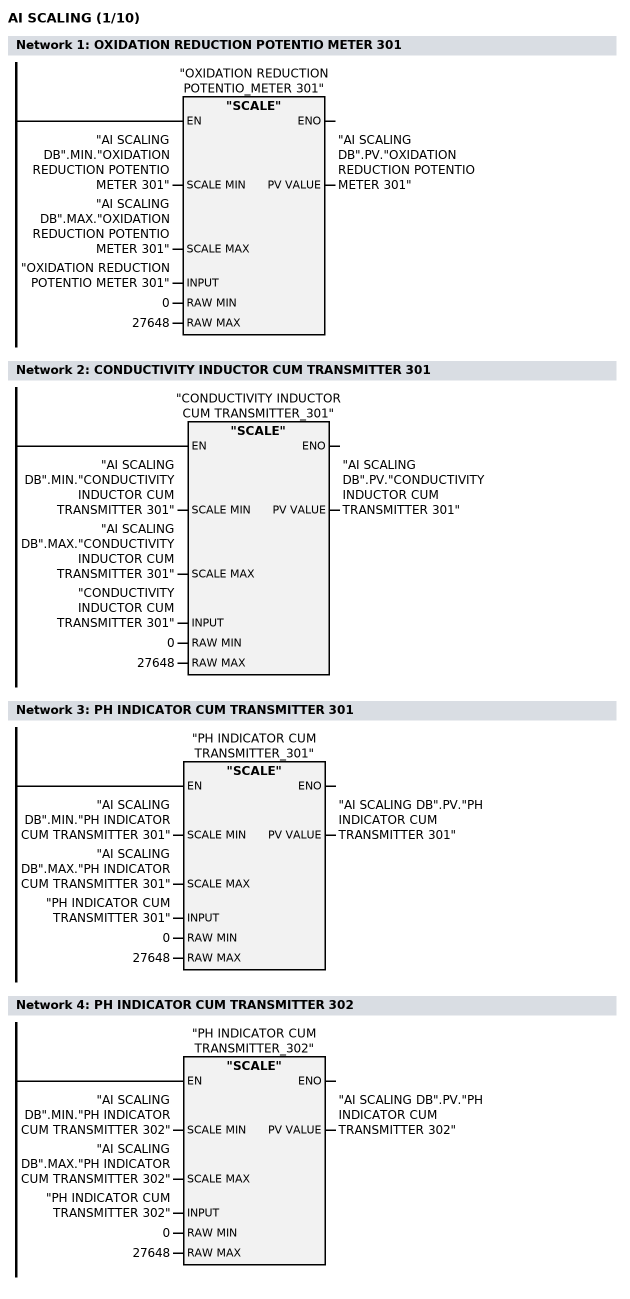
   RUNG wire#powerrail
      "OXIDATION REDUCTION POTENTIO_METER 301"("SCALE MIN" := "AI SCALING DB".MIN."OXIDATION REDUCTION POTENTIO METER 301", "SCALE MAX" := "AI SCALING DB".MAX."OXIDATION REDUCTION POTENTIO METER 301", INPUT := "OXIDATION REDUCTION POTENTIO METER 301", "RAW MIN" := 0, "RAW MAX" := 27648, "PV VALUE" => "AI SCALING DB".PV."OXIDATION REDUCTION POTENTIO METER 301")
   END_RUNG
   // the same network as SCL:
   "OXIDATION REDUCTION POTENTIO_METER 301"("SCALE MIN" := "AI SCALING DB".MIN."OXIDATION REDUCTION POTENTIO METER 301",   // "SCALE"
                           "SCALE MAX" := "AI SCALING DB".MAX."OXIDATION REDUCTION POTENTIO METER 301",
                           INPUT := "OXIDATION REDUCTION POTENTIO METER 301",
                           "RAW MIN" := 0,
                           "RAW MAX" := 27648,
                           "PV VALUE" => "AI SCALING DB".PV."OXIDATION REDUCTION POTENTIO METER 301");
END_REGION

REGION Network 2: CONDUCTIVITY INDUCTOR CUM TRANSMITTER 301
   RUNG wire#powerrail
      "CONDUCTIVITY INDUCTOR CUM TRANSMITTER_301"("SCALE MIN" := "AI SCALING DB".MIN."CONDUCTIVITY INDUCTOR CUM TRANSMITTER 301", "SCALE MAX" := "AI SCALING DB".MAX."CONDUCTIVITY INDUCTOR CUM TRANSMITTER 301", INPUT := "CONDUCTIVITY INDUCTOR CUM TRANSMITTER 301", "RAW MIN" := 0, "RAW MAX" := 27648, "PV VALUE" => "AI SCALING DB".PV."CONDUCTIVITY INDUCTOR CUM TRANSMITTER 301")
   END_RUNG
   // the same network as SCL:
   "CONDUCTIVITY INDUCTOR CUM TRANSMITTER_301"("SCALE MIN" := "AI SCALING DB".MIN."CONDUCTIVITY INDUCTOR CUM TRANSMITTER 301",   // "SCALE"
                           "SCALE MAX" := "AI SCALING DB".MAX."CONDUCTIVITY INDUCTOR CUM TRANSMITTER 301",
                           INPUT := "CONDUCTIVITY INDUCTOR CUM TRANSMITTER 301",
                           "RAW MIN" := 0,
                           "RAW MAX" := 27648,
                           "PV VALUE" => "AI SCALING DB".PV."CONDUCTIVITY INDUCTOR CUM TRANSMITTER 301");
END_REGION

REGION Network 3: PH INDICATOR CUM TRANSMITTER 301
   RUNG wire#powerrail
      "PH INDICATOR CUM TRANSMITTER_301"("SCALE MIN" := "AI SCALING DB".MIN."PH INDICATOR CUM TRANSMITTER 301", "SCALE MAX" := "AI SCALING DB".MAX."PH INDICATOR CUM TRANSMITTER 301", INPUT := "PH INDICATOR CUM TRANSMITTER 301", "RAW MIN" := 0, "RAW MAX" := 27648, "PV VALUE" => "AI SCALING DB".PV."PH INDICATOR CUM TRANSMITTER 301")
   END_RUNG
   // the same network as SCL:
   "PH INDICATOR CUM TRANSMITTER_301"("SCALE MIN" := "AI SCALING DB".MIN."PH INDICATOR CUM TRANSMITTER 301",   // "SCALE"
                           "SCALE MAX" := "AI SCALING DB".MAX."PH INDICATOR CUM TRANSMITTER 301",
                           INPUT := "PH INDICATOR CUM TRANSMITTER 301",
                           "RAW MIN" := 0,
                           "RAW MAX" := 27648,
                           "PV VALUE" => "AI SCALING DB".PV."PH INDICATOR CUM TRANSMITTER 301");
END_REGION

REGION Network 4: PH INDICATOR CUM TRANSMITTER 302
   RUNG wire#powerrail
      "PH INDICATOR CUM TRANSMITTER_302"("SCALE MIN" := "AI SCALING DB".MIN."PH INDICATOR CUM TRANSMITTER 302", "SCALE MAX" := "AI SCALING DB".MAX."PH INDICATOR CUM TRANSMITTER 302", INPUT := "PH INDICATOR CUM TRANSMITTER 302", "RAW MIN" := 0, "RAW MAX" := 27648, "PV VALUE" => "AI SCALING DB".PV."PH INDICATOR CUM TRANSMITTER 302")
   END_RUNG
   // the same network as SCL:
   "PH INDICATOR CUM TRANSMITTER_302"("SCALE MIN" := "AI SCALING DB".MIN."PH INDICATOR CUM TRANSMITTER 302",   // "SCALE"
                           "SCALE MAX" := "AI SCALING DB".MAX."PH INDICATOR CUM TRANSMITTER 302",
                           INPUT := "PH INDICATOR CUM TRANSMITTER 302",
                           "RAW MIN" := 0,
                           "RAW MAX" := 27648,
                           "PV VALUE" => "AI SCALING DB".PV."PH INDICATOR CUM TRANSMITTER 302");
END_REGION

REGION Network 5: CONDUCTIVITY INDICATOR CUM TRANSMITTER 302
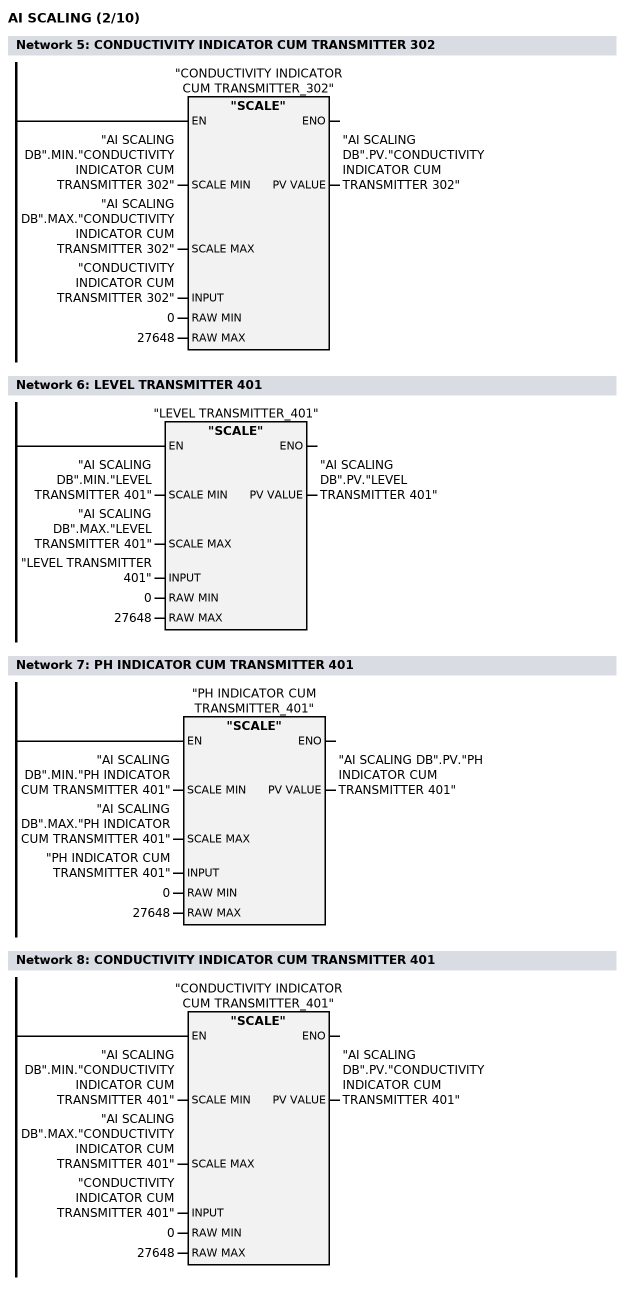
   RUNG wire#powerrail
      "CONDUCTIVITY INDICATOR CUM TRANSMITTER_302"("SCALE MIN" := "AI SCALING DB".MIN."CONDUCTIVITY INDICATOR CUM TRANSMITTER 302", "SCALE MAX" := "AI SCALING DB".MAX."CONDUCTIVITY INDICATOR CUM TRANSMITTER 302", INPUT := "CONDUCTIVITY INDICATOR CUM TRANSMITTER 302", "RAW MIN" := 0, "RAW MAX" := 27648, "PV VALUE" => "AI SCALING DB".PV."CONDUCTIVITY INDICATOR CUM TRANSMITTER 302")
   END_RUNG
   // the same network as SCL:
   "CONDUCTIVITY INDICATOR CUM TRANSMITTER_302"("SCALE MIN" := "AI SCALING DB".MIN."CONDUCTIVITY INDICATOR CUM TRANSMITTER 302",   // "SCALE"
                           "SCALE MAX" := "AI SCALING DB".MAX."CONDUCTIVITY INDICATOR CUM TRANSMITTER 302",
                           INPUT := "CONDUCTIVITY INDICATOR CUM TRANSMITTER 302",
                           "RAW MIN" := 0,
                           "RAW MAX" := 27648,
                           "PV VALUE" => "AI SCALING DB".PV."CONDUCTIVITY INDICATOR CUM TRANSMITTER 302");
END_REGION

REGION Network 6: LEVEL TRANSMITTER 401
   RUNG wire#powerrail
      "LEVEL TRANSMITTER_401"("SCALE MIN" := "AI SCALING DB".MIN."LEVEL TRANSMITTER 401", "SCALE MAX" := "AI SCALING DB".MAX."LEVEL TRANSMITTER 401", INPUT := "LEVEL TRANSMITTER 401", "RAW MIN" := 0, "RAW MAX" := 27648, "PV VALUE" => "AI SCALING DB".PV."LEVEL TRANSMITTER 401")
   END_RUNG
   // the same network as SCL:
   "LEVEL TRANSMITTER_401"("SCALE MIN" := "AI SCALING DB".MIN."LEVEL TRANSMITTER 401",   // "SCALE"
                           "SCALE MAX" := "AI SCALING DB".MAX."LEVEL TRANSMITTER 401",
                           INPUT := "LEVEL TRANSMITTER 401",
                           "RAW MIN" := 0,
                           "RAW MAX" := 27648,
                           "PV VALUE" => "AI SCALING DB".PV."LEVEL TRANSMITTER 401");
END_REGION

REGION Network 7: PH INDICATOR CUM TRANSMITTER 401
   RUNG wire#powerrail
      "PH INDICATOR CUM TRANSMITTER_401"("SCALE MIN" := "AI SCALING DB".MIN."PH INDICATOR CUM TRANSMITTER 401", "SCALE MAX" := "AI SCALING DB".MAX."PH INDICATOR CUM TRANSMITTER 401", INPUT := "PH INDICATOR CUM TRANSMITTER 401", "RAW MIN" := 0, "RAW MAX" := 27648, "PV VALUE" => "AI SCALING DB".PV."PH INDICATOR CUM TRANSMITTER 401")
   END_RUNG
   // the same network as SCL:
   "PH INDICATOR CUM TRANSMITTER_401"("SCALE MIN" := "AI SCALING DB".MIN."PH INDICATOR CUM TRANSMITTER 401",   // "SCALE"
                           "SCALE MAX" := "AI SCALING DB".MAX."PH INDICATOR CUM TRANSMITTER 401",
                           INPUT := "PH INDICATOR CUM TRANSMITTER 401",
                           "RAW MIN" := 0,
                           "RAW MAX" := 27648,
                           "PV VALUE" => "AI SCALING DB".PV."PH INDICATOR CUM TRANSMITTER 401");
END_REGION

REGION Network 8: CONDUCTIVITY INDICATOR CUM TRANSMITTER 401
   RUNG wire#powerrail
      "CONDUCTIVITY INDICATOR CUM TRANSMITTER_401"("SCALE MIN" := "AI SCALING DB".MIN."CONDUCTIVITY INDICATOR CUM TRANSMITTER 401", "SCALE MAX" := "AI SCALING DB".MAX."CONDUCTIVITY INDICATOR CUM TRANSMITTER 401", INPUT := "CONDUCTIVITY INDICATOR CUM TRANSMITTER 401", "RAW MIN" := 0, "RAW MAX" := 27648, "PV VALUE" => "AI SCALING DB".PV."CONDUCTIVITY INDICATOR CUM TRANSMITTER 401")
   END_RUNG
   // the same network as SCL:
   "CONDUCTIVITY INDICATOR CUM TRANSMITTER_401"("SCALE MIN" := "AI SCALING DB".MIN."CONDUCTIVITY INDICATOR CUM TRANSMITTER 401",   // "SCALE"
                           "SCALE MAX" := "AI SCALING DB".MAX."CONDUCTIVITY INDICATOR CUM TRANSMITTER 401",
                           INPUT := "CONDUCTIVITY INDICATOR CUM TRANSMITTER 401",
                           "RAW MIN" := 0,
                           "RAW MAX" := 27648,
                           "PV VALUE" => "AI SCALING DB".PV."CONDUCTIVITY INDICATOR CUM TRANSMITTER 401");
END_REGION

REGION Network 9: CONFUCTIVITY INDICATOR CUM TRANSMITTER 402
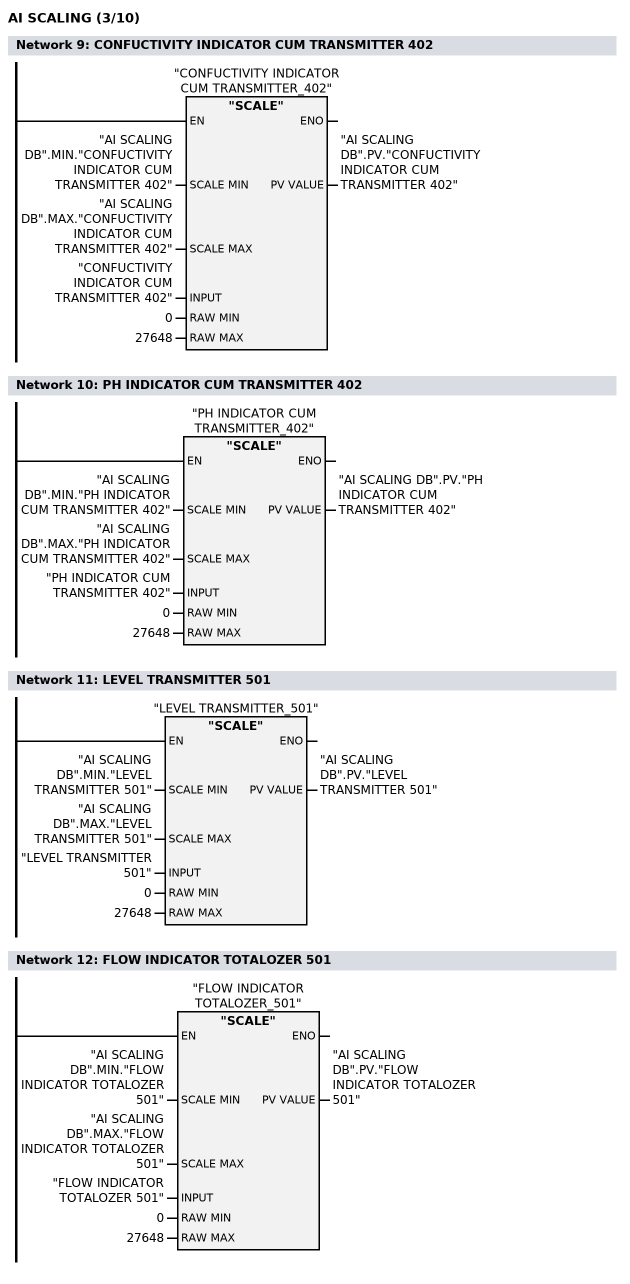
   RUNG wire#powerrail
      "CONFUCTIVITY INDICATOR CUM TRANSMITTER_402"("SCALE MIN" := "AI SCALING DB".MIN."CONFUCTIVITY INDICATOR CUM TRANSMITTER 402", "SCALE MAX" := "AI SCALING DB".MAX."CONFUCTIVITY INDICATOR CUM TRANSMITTER 402", INPUT := "CONFUCTIVITY INDICATOR CUM TRANSMITTER 402", "RAW MIN" := 0, "RAW MAX" := 27648, "PV VALUE" => "AI SCALING DB".PV."CONFUCTIVITY INDICATOR CUM TRANSMITTER 402")
   END_RUNG
   // the same network as SCL:
   "CONFUCTIVITY INDICATOR CUM TRANSMITTER_402"("SCALE MIN" := "AI SCALING DB".MIN."CONFUCTIVITY INDICATOR CUM TRANSMITTER 402",   // "SCALE"
                           "SCALE MAX" := "AI SCALING DB".MAX."CONFUCTIVITY INDICATOR CUM TRANSMITTER 402",
                           INPUT := "CONFUCTIVITY INDICATOR CUM TRANSMITTER 402",
                           "RAW MIN" := 0,
                           "RAW MAX" := 27648,
                           "PV VALUE" => "AI SCALING DB".PV."CONFUCTIVITY INDICATOR CUM TRANSMITTER 402");
END_REGION

REGION Network 10: PH INDICATOR CUM TRANSMITTER 402
   RUNG wire#powerrail
      "PH INDICATOR CUM TRANSMITTER_402"("SCALE MIN" := "AI SCALING DB".MIN."PH INDICATOR CUM TRANSMITTER 402", "SCALE MAX" := "AI SCALING DB".MAX."PH INDICATOR CUM TRANSMITTER 402", INPUT := "PH INDICATOR CUM TRANSMITTER 402", "RAW MIN" := 0, "RAW MAX" := 27648, "PV VALUE" => "AI SCALING DB".PV."PH INDICATOR CUM TRANSMITTER 402")
   END_RUNG
   // the same network as SCL:
   "PH INDICATOR CUM TRANSMITTER_402"("SCALE MIN" := "AI SCALING DB".MIN."PH INDICATOR CUM TRANSMITTER 402",   // "SCALE"
                           "SCALE MAX" := "AI SCALING DB".MAX."PH INDICATOR CUM TRANSMITTER 402",
                           INPUT := "PH INDICATOR CUM TRANSMITTER 402",
                           "RAW MIN" := 0,
                           "RAW MAX" := 27648,
                           "PV VALUE" => "AI SCALING DB".PV."PH INDICATOR CUM TRANSMITTER 402");
END_REGION

REGION Network 11: LEVEL TRANSMITTER 501
   RUNG wire#powerrail
      "LEVEL TRANSMITTER_501"("SCALE MIN" := "AI SCALING DB".MIN."LEVEL TRANSMITTER 501", "SCALE MAX" := "AI SCALING DB".MAX."LEVEL TRANSMITTER 501", INPUT := "LEVEL TRANSMITTER 501", "RAW MIN" := 0, "RAW MAX" := 27648, "PV VALUE" => "AI SCALING DB".PV."LEVEL TRANSMITTER 501")
   END_RUNG
   // the same network as SCL:
   "LEVEL TRANSMITTER_501"("SCALE MIN" := "AI SCALING DB".MIN."LEVEL TRANSMITTER 501",   // "SCALE"
                           "SCALE MAX" := "AI SCALING DB".MAX."LEVEL TRANSMITTER 501",
                           INPUT := "LEVEL TRANSMITTER 501",
                           "RAW MIN" := 0,
                           "RAW MAX" := 27648,
                           "PV VALUE" => "AI SCALING DB".PV."LEVEL TRANSMITTER 501");
END_REGION

REGION Network 12: FLOW INDICATOR TOTALOZER 501
   RUNG wire#powerrail
      "FLOW INDICATOR TOTALOZER_501"("SCALE MIN" := "AI SCALING DB".MIN."FLOW INDICATOR TOTALOZER 501", "SCALE MAX" := "AI SCALING DB".MAX."FLOW INDICATOR TOTALOZER 501", INPUT := "FLOW INDICATOR TOTALOZER 501", "RAW MIN" := 0, "RAW MAX" := 27648, "PV VALUE" => "AI SCALING DB".PV."FLOW INDICATOR TOTALOZER 501")
   END_RUNG
   // the same network as SCL:
   "FLOW INDICATOR TOTALOZER_501"("SCALE MIN" := "AI SCALING DB".MIN."FLOW INDICATOR TOTALOZER 501",   // "SCALE"
                           "SCALE MAX" := "AI SCALING DB".MAX."FLOW INDICATOR TOTALOZER 501",
                           INPUT := "FLOW INDICATOR TOTALOZER 501",
                           "RAW MIN" := 0,
                           "RAW MAX" := 27648,
                           "PV VALUE" => "AI SCALING DB".PV."FLOW INDICATOR TOTALOZER 501");
END_REGION

REGION Network 13: PRESSURE TRANSMITTER 501
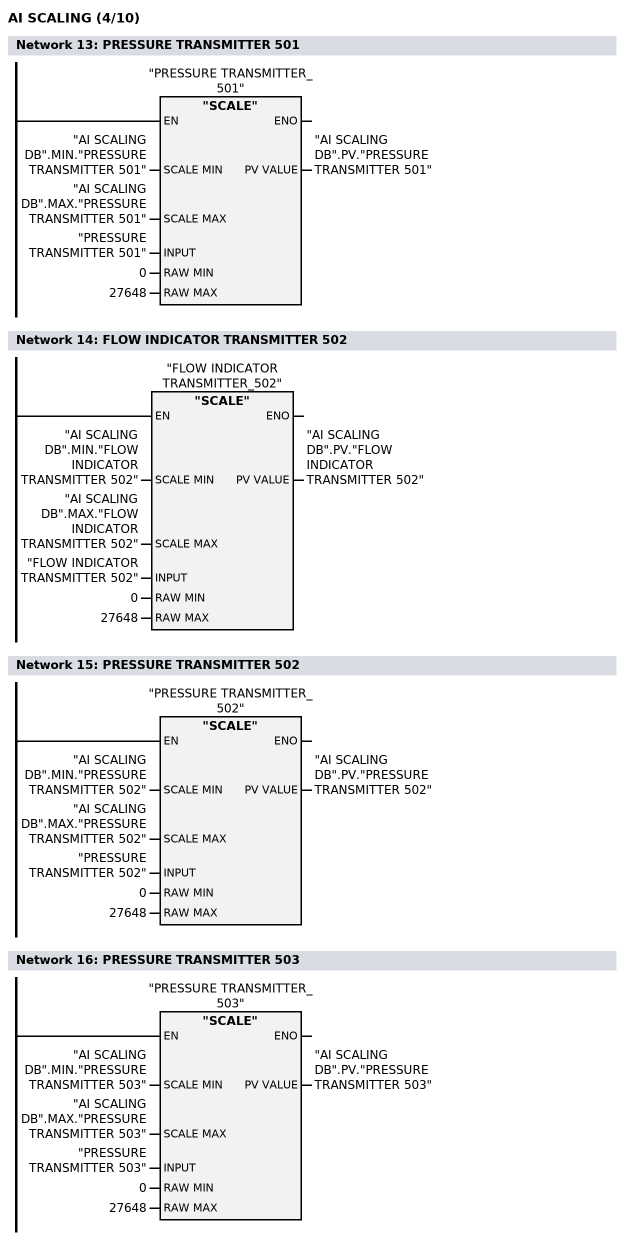
   RUNG wire#powerrail
      "PRESSURE TRANSMITTER_501"("SCALE MIN" := "AI SCALING DB".MIN."PRESSURE TRANSMITTER 501", "SCALE MAX" := "AI SCALING DB".MAX."PRESSURE TRANSMITTER 501", INPUT := "PRESSURE TRANSMITTER 501", "RAW MIN" := 0, "RAW MAX" := 27648, "PV VALUE" => "AI SCALING DB".PV."PRESSURE TRANSMITTER 501")
   END_RUNG
   // the same network as SCL:
   "PRESSURE TRANSMITTER_501"("SCALE MIN" := "AI SCALING DB".MIN."PRESSURE TRANSMITTER 501",   // "SCALE"
                           "SCALE MAX" := "AI SCALING DB".MAX."PRESSURE TRANSMITTER 501",
                           INPUT := "PRESSURE TRANSMITTER 501",
                           "RAW MIN" := 0,
                           "RAW MAX" := 27648,
                           "PV VALUE" => "AI SCALING DB".PV."PRESSURE TRANSMITTER 501");
END_REGION

REGION Network 14: FLOW INDICATOR TRANSMITTER 502
   RUNG wire#powerrail
      "FLOW INDICATOR TRANSMITTER_502"("SCALE MIN" := "AI SCALING DB".MIN."FLOW INDICATOR TRANSMITTER 502", "SCALE MAX" := "AI SCALING DB".MAX."FLOW INDICATOR TRANSMITTER 502", INPUT := "FLOW INDICATOR TRANSMITTER 502", "RAW MIN" := 0, "RAW MAX" := 27648, "PV VALUE" => "AI SCALING DB".PV."FLOW INDICATOR TRANSMITTER 502")
   END_RUNG
   // the same network as SCL:
   "FLOW INDICATOR TRANSMITTER_502"("SCALE MIN" := "AI SCALING DB".MIN."FLOW INDICATOR TRANSMITTER 502",   // "SCALE"
                           "SCALE MAX" := "AI SCALING DB".MAX."FLOW INDICATOR TRANSMITTER 502",
                           INPUT := "FLOW INDICATOR TRANSMITTER 502",
                           "RAW MIN" := 0,
                           "RAW MAX" := 27648,
                           "PV VALUE" => "AI SCALING DB".PV."FLOW INDICATOR TRANSMITTER 502");
END_REGION

REGION Network 15: PRESSURE TRANSMITTER 502
   RUNG wire#powerrail
      "PRESSURE TRANSMITTER_502"("SCALE MIN" := "AI SCALING DB".MIN."PRESSURE TRANSMITTER 502", "SCALE MAX" := "AI SCALING DB".MAX."PRESSURE TRANSMITTER 502", INPUT := "PRESSURE TRANSMITTER 502", "RAW MIN" := 0, "RAW MAX" := 27648, "PV VALUE" => "AI SCALING DB".PV."PRESSURE TRANSMITTER 502")
   END_RUNG
   // the same network as SCL:
   "PRESSURE TRANSMITTER_502"("SCALE MIN" := "AI SCALING DB".MIN."PRESSURE TRANSMITTER 502",   // "SCALE"
                           "SCALE MAX" := "AI SCALING DB".MAX."PRESSURE TRANSMITTER 502",
                           INPUT := "PRESSURE TRANSMITTER 502",
                           "RAW MIN" := 0,
                           "RAW MAX" := 27648,
                           "PV VALUE" => "AI SCALING DB".PV."PRESSURE TRANSMITTER 502");
END_REGION

REGION Network 16: PRESSURE TRANSMITTER 503
   RUNG wire#powerrail
      "PRESSURE TRANSMITTER_503"("SCALE MIN" := "AI SCALING DB".MIN."PRESSURE TRANSMITTER 503", "SCALE MAX" := "AI SCALING DB".MAX."PRESSURE TRANSMITTER 503", INPUT := "PRESSURE TRANSMITTER 503", "RAW MIN" := 0, "RAW MAX" := 27648, "PV VALUE" => "AI SCALING DB".PV."PRESSURE TRANSMITTER 503")
   END_RUNG
   // the same network as SCL:
   "PRESSURE TRANSMITTER_503"("SCALE MIN" := "AI SCALING DB".MIN."PRESSURE TRANSMITTER 503",   // "SCALE"
                           "SCALE MAX" := "AI SCALING DB".MAX."PRESSURE TRANSMITTER 503",
                           INPUT := "PRESSURE TRANSMITTER 503",
                           "RAW MIN" := 0,
                           "RAW MAX" := 27648,
                           "PV VALUE" => "AI SCALING DB".PV."PRESSURE TRANSMITTER 503");
END_REGION

REGION Network 17: PRESSURE TRANSMITTER 504
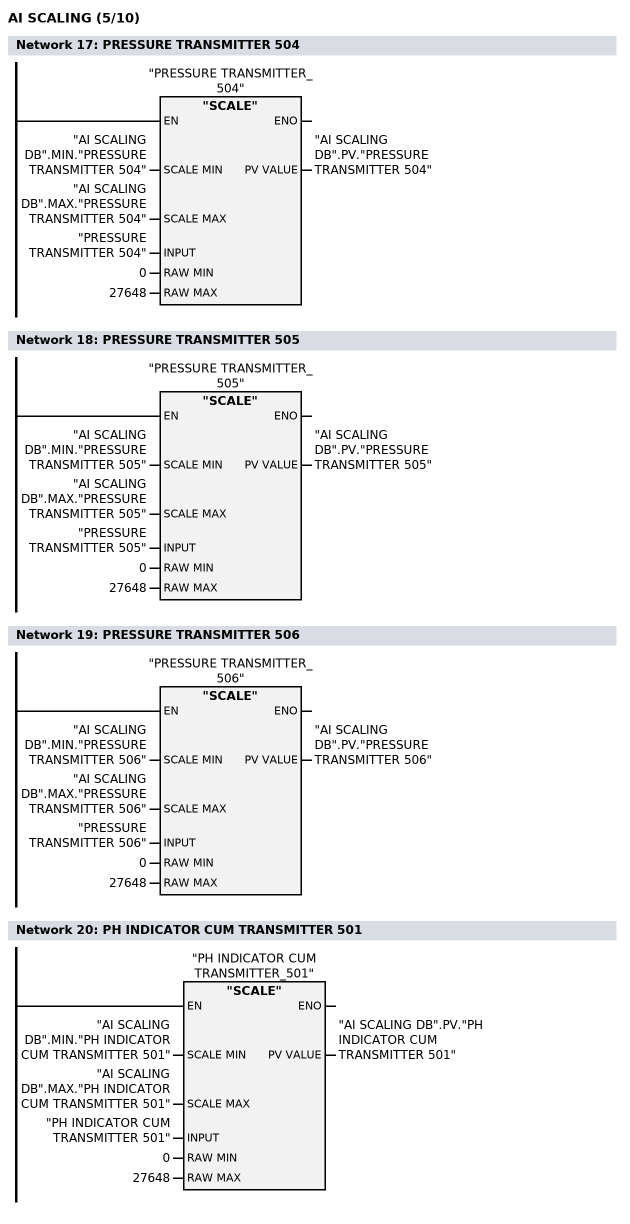
   RUNG wire#powerrail
      "PRESSURE TRANSMITTER_504"("SCALE MIN" := "AI SCALING DB".MIN."PRESSURE TRANSMITTER 504", "SCALE MAX" := "AI SCALING DB".MAX."PRESSURE TRANSMITTER 504", INPUT := "PRESSURE TRANSMITTER 504", "RAW MIN" := 0, "RAW MAX" := 27648, "PV VALUE" => "AI SCALING DB".PV."PRESSURE TRANSMITTER 504")
   END_RUNG
   // the same network as SCL:
   "PRESSURE TRANSMITTER_504"("SCALE MIN" := "AI SCALING DB".MIN."PRESSURE TRANSMITTER 504",   // "SCALE"
                           "SCALE MAX" := "AI SCALING DB".MAX."PRESSURE TRANSMITTER 504",
                           INPUT := "PRESSURE TRANSMITTER 504",
                           "RAW MIN" := 0,
                           "RAW MAX" := 27648,
                           "PV VALUE" => "AI SCALING DB".PV."PRESSURE TRANSMITTER 504");
END_REGION

REGION Network 18: PRESSURE TRANSMITTER 505
   RUNG wire#powerrail
      "PRESSURE TRANSMITTER_505"("SCALE MIN" := "AI SCALING DB".MIN."PRESSURE TRANSMITTER 505", "SCALE MAX" := "AI SCALING DB".MAX."PRESSURE TRANSMITTER 505", INPUT := "PRESSURE TRANSMITTER 505", "RAW MIN" := 0, "RAW MAX" := 27648, "PV VALUE" => "AI SCALING DB".PV."PRESSURE TRANSMITTER 505")
   END_RUNG
   // the same network as SCL:
   "PRESSURE TRANSMITTER_505"("SCALE MIN" := "AI SCALING DB".MIN."PRESSURE TRANSMITTER 505",   // "SCALE"
                           "SCALE MAX" := "AI SCALING DB".MAX."PRESSURE TRANSMITTER 505",
                           INPUT := "PRESSURE TRANSMITTER 505",
                           "RAW MIN" := 0,
                           "RAW MAX" := 27648,
                           "PV VALUE" => "AI SCALING DB".PV."PRESSURE TRANSMITTER 505");
END_REGION

REGION Network 19: PRESSURE TRANSMITTER 506
   RUNG wire#powerrail
      "PRESSURE TRANSMITTER_506"("SCALE MIN" := "AI SCALING DB".MIN."PRESSURE TRANSMITTER 506", "SCALE MAX" := "AI SCALING DB".MAX."PRESSURE TRANSMITTER 506", INPUT := "PRESSURE TRANSMITTER 506", "RAW MIN" := 0, "RAW MAX" := 27648, "PV VALUE" => "AI SCALING DB".PV."PRESSURE TRANSMITTER 506")
   END_RUNG
   // the same network as SCL:
   "PRESSURE TRANSMITTER_506"("SCALE MIN" := "AI SCALING DB".MIN."PRESSURE TRANSMITTER 506",   // "SCALE"
                           "SCALE MAX" := "AI SCALING DB".MAX."PRESSURE TRANSMITTER 506",
                           INPUT := "PRESSURE TRANSMITTER 506",
                           "RAW MIN" := 0,
                           "RAW MAX" := 27648,
                           "PV VALUE" => "AI SCALING DB".PV."PRESSURE TRANSMITTER 506");
END_REGION

REGION Network 20: PH INDICATOR CUM TRANSMITTER 501
   RUNG wire#powerrail
      "PH INDICATOR CUM TRANSMITTER_501"("SCALE MIN" := "AI SCALING DB".MIN."PH INDICATOR CUM TRANSMITTER 501", "SCALE MAX" := "AI SCALING DB".MAX."PH INDICATOR CUM TRANSMITTER 501", INPUT := "PH INDICATOR CUM TRANSMITTER 501", "RAW MIN" := 0, "RAW MAX" := 27648, "PV VALUE" => "AI SCALING DB".PV."PH INDICATOR CUM TRANSMITTER 501")
   END_RUNG
   // the same network as SCL:
   "PH INDICATOR CUM TRANSMITTER_501"("SCALE MIN" := "AI SCALING DB".MIN."PH INDICATOR CUM TRANSMITTER 501",   // "SCALE"
                           "SCALE MAX" := "AI SCALING DB".MAX."PH INDICATOR CUM TRANSMITTER 501",
                           INPUT := "PH INDICATOR CUM TRANSMITTER 501",
                           "RAW MIN" := 0,
                           "RAW MAX" := 27648,
                           "PV VALUE" => "AI SCALING DB".PV."PH INDICATOR CUM TRANSMITTER 501");
END_REGION

REGION Network 21: PH INDICATOR CUM TRANSMITTER 502
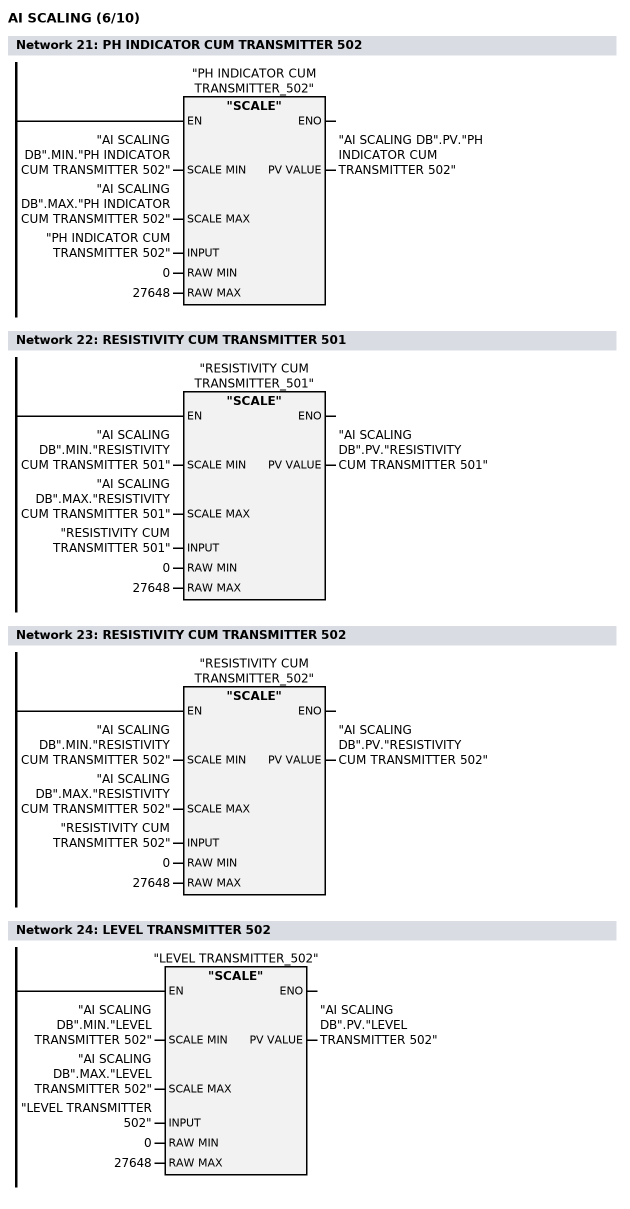
   RUNG wire#powerrail
      "PH INDICATOR CUM TRANSMITTER_502"("SCALE MIN" := "AI SCALING DB".MIN."PH INDICATOR CUM TRANSMITTER 502", "SCALE MAX" := "AI SCALING DB".MAX."PH INDICATOR CUM TRANSMITTER 502", INPUT := "PH INDICATOR CUM TRANSMITTER 502", "RAW MIN" := 0, "RAW MAX" := 27648, "PV VALUE" => "AI SCALING DB".PV."PH INDICATOR CUM TRANSMITTER 502")
   END_RUNG
   // the same network as SCL:
   "PH INDICATOR CUM TRANSMITTER_502"("SCALE MIN" := "AI SCALING DB".MIN."PH INDICATOR CUM TRANSMITTER 502",   // "SCALE"
                           "SCALE MAX" := "AI SCALING DB".MAX."PH INDICATOR CUM TRANSMITTER 502",
                           INPUT := "PH INDICATOR CUM TRANSMITTER 502",
                           "RAW MIN" := 0,
                           "RAW MAX" := 27648,
                           "PV VALUE" => "AI SCALING DB".PV."PH INDICATOR CUM TRANSMITTER 502");
END_REGION

REGION Network 22: RESISTIVITY CUM TRANSMITTER 501
   RUNG wire#powerrail
      "RESISTIVITY CUM TRANSMITTER_501"("SCALE MIN" := "AI SCALING DB".MIN."RESISTIVITY CUM TRANSMITTER 501", "SCALE MAX" := "AI SCALING DB".MAX."RESISTIVITY CUM TRANSMITTER 501", INPUT := "RESISTIVITY CUM TRANSMITTER 501", "RAW MIN" := 0, "RAW MAX" := 27648, "PV VALUE" => "AI SCALING DB".PV."RESISTIVITY CUM TRANSMITTER 501")
   END_RUNG
   // the same network as SCL:
   "RESISTIVITY CUM TRANSMITTER_501"("SCALE MIN" := "AI SCALING DB".MIN."RESISTIVITY CUM TRANSMITTER 501",   // "SCALE"
                           "SCALE MAX" := "AI SCALING DB".MAX."RESISTIVITY CUM TRANSMITTER 501",
                           INPUT := "RESISTIVITY CUM TRANSMITTER 501",
                           "RAW MIN" := 0,
                           "RAW MAX" := 27648,
                           "PV VALUE" => "AI SCALING DB".PV."RESISTIVITY CUM TRANSMITTER 501");
END_REGION

REGION Network 23: RESISTIVITY CUM TRANSMITTER 502
   RUNG wire#powerrail
      "RESISTIVITY CUM TRANSMITTER_502"("SCALE MIN" := "AI SCALING DB".MIN."RESISTIVITY CUM TRANSMITTER 502", "SCALE MAX" := "AI SCALING DB".MAX."RESISTIVITY CUM TRANSMITTER 502", INPUT := "RESISTIVITY CUM TRANSMITTER 502", "RAW MIN" := 0, "RAW MAX" := 27648, "PV VALUE" => "AI SCALING DB".PV."RESISTIVITY CUM TRANSMITTER 502")
   END_RUNG
   // the same network as SCL:
   "RESISTIVITY CUM TRANSMITTER_502"("SCALE MIN" := "AI SCALING DB".MIN."RESISTIVITY CUM TRANSMITTER 502",   // "SCALE"
                           "SCALE MAX" := "AI SCALING DB".MAX."RESISTIVITY CUM TRANSMITTER 502",
                           INPUT := "RESISTIVITY CUM TRANSMITTER 502",
                           "RAW MIN" := 0,
                           "RAW MAX" := 27648,
                           "PV VALUE" => "AI SCALING DB".PV."RESISTIVITY CUM TRANSMITTER 502");
END_REGION

REGION Network 24: LEVEL TRANSMITTER 502
   RUNG wire#powerrail
      "LEVEL TRANSMITTER_502"("SCALE MIN" := "AI SCALING DB".MIN."LEVEL TRANSMITTER 502", "SCALE MAX" := "AI SCALING DB".MAX."LEVEL TRANSMITTER 502", INPUT := "LEVEL TRANSMITTER 502", "RAW MIN" := 0, "RAW MAX" := 27648, "PV VALUE" => "AI SCALING DB".PV."LEVEL TRANSMITTER 502")
   END_RUNG
   // the same network as SCL:
   "LEVEL TRANSMITTER_502"("SCALE MIN" := "AI SCALING DB".MIN."LEVEL TRANSMITTER 502",   // "SCALE"
                           "SCALE MAX" := "AI SCALING DB".MAX."LEVEL TRANSMITTER 502",
                           INPUT := "LEVEL TRANSMITTER 502",
                           "RAW MIN" := 0,
                           "RAW MAX" := 27648,
                           "PV VALUE" => "AI SCALING DB".PV."LEVEL TRANSMITTER 502");
END_REGION

REGION Network 25: FLOW INDICATOR TRANSMITTER 503
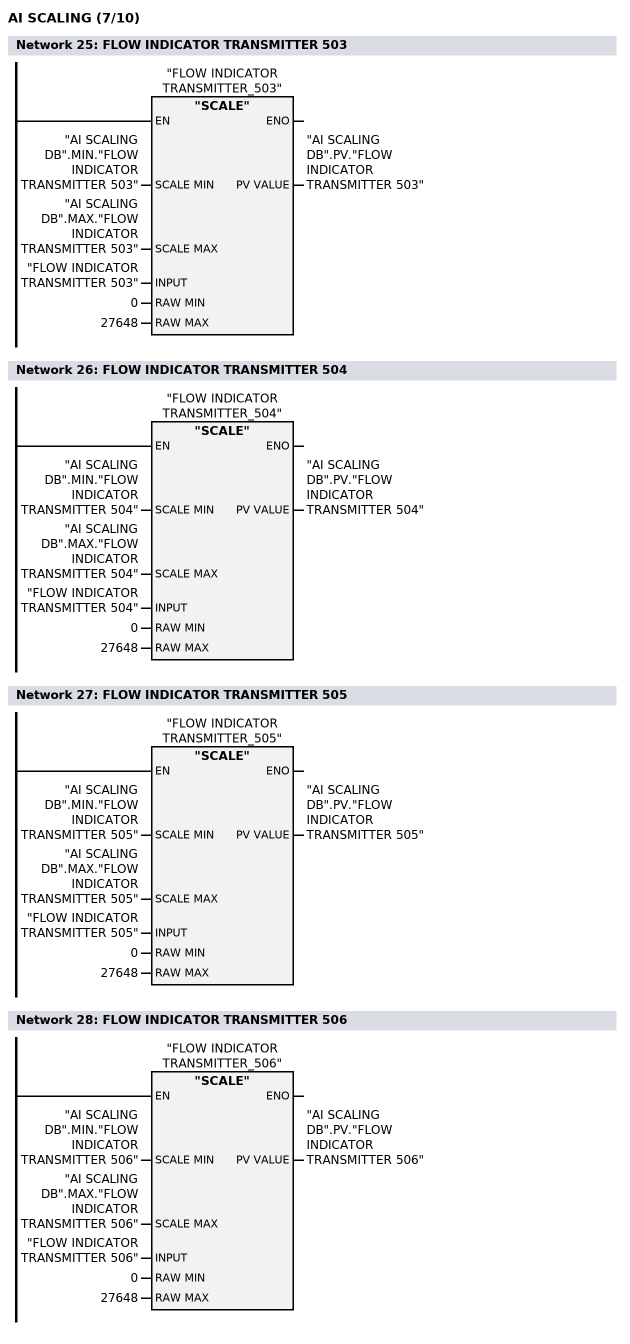
   RUNG wire#powerrail
      "FLOW INDICATOR TRANSMITTER_503"("SCALE MIN" := "AI SCALING DB".MIN."FLOW INDICATOR TRANSMITTER 503", "SCALE MAX" := "AI SCALING DB".MAX."FLOW INDICATOR TRANSMITTER 503", INPUT := "FLOW INDICATOR TRANSMITTER 503", "RAW MIN" := 0, "RAW MAX" := 27648, "PV VALUE" => "AI SCALING DB".PV."FLOW INDICATOR TRANSMITTER 503")
   END_RUNG
   // the same network as SCL:
   "FLOW INDICATOR TRANSMITTER_503"("SCALE MIN" := "AI SCALING DB".MIN."FLOW INDICATOR TRANSMITTER 503",   // "SCALE"
                           "SCALE MAX" := "AI SCALING DB".MAX."FLOW INDICATOR TRANSMITTER 503",
                           INPUT := "FLOW INDICATOR TRANSMITTER 503",
                           "RAW MIN" := 0,
                           "RAW MAX" := 27648,
                           "PV VALUE" => "AI SCALING DB".PV."FLOW INDICATOR TRANSMITTER 503");
END_REGION

REGION Network 26: FLOW INDICATOR TRANSMITTER 504
   RUNG wire#powerrail
      "FLOW INDICATOR TRANSMITTER_504"("SCALE MIN" := "AI SCALING DB".MIN."FLOW INDICATOR TRANSMITTER 504", "SCALE MAX" := "AI SCALING DB".MAX."FLOW INDICATOR TRANSMITTER 504", INPUT := "FLOW INDICATOR TRANSMITTER 504", "RAW MIN" := 0, "RAW MAX" := 27648, "PV VALUE" => "AI SCALING DB".PV."FLOW INDICATOR TRANSMITTER 504")
   END_RUNG
   // the same network as SCL:
   "FLOW INDICATOR TRANSMITTER_504"("SCALE MIN" := "AI SCALING DB".MIN."FLOW INDICATOR TRANSMITTER 504",   // "SCALE"
                           "SCALE MAX" := "AI SCALING DB".MAX."FLOW INDICATOR TRANSMITTER 504",
                           INPUT := "FLOW INDICATOR TRANSMITTER 504",
                           "RAW MIN" := 0,
                           "RAW MAX" := 27648,
                           "PV VALUE" => "AI SCALING DB".PV."FLOW INDICATOR TRANSMITTER 504");
END_REGION

REGION Network 27: FLOW INDICATOR TRANSMITTER 505
   RUNG wire#powerrail
      "FLOW INDICATOR TRANSMITTER_505"("SCALE MIN" := "AI SCALING DB".MIN."FLOW INDICATOR TRANSMITTER 505", "SCALE MAX" := "AI SCALING DB".MAX."FLOW INDICATOR TRANSMITTER 505", INPUT := "FLOW INDICATOR TRANSMITTER 505", "RAW MIN" := 0, "RAW MAX" := 27648, "PV VALUE" => "AI SCALING DB".PV."FLOW INDICATOR TRANSMITTER 505")
   END_RUNG
   // the same network as SCL:
   "FLOW INDICATOR TRANSMITTER_505"("SCALE MIN" := "AI SCALING DB".MIN."FLOW INDICATOR TRANSMITTER 505",   // "SCALE"
                           "SCALE MAX" := "AI SCALING DB".MAX."FLOW INDICATOR TRANSMITTER 505",
                           INPUT := "FLOW INDICATOR TRANSMITTER 505",
                           "RAW MIN" := 0,
                           "RAW MAX" := 27648,
                           "PV VALUE" => "AI SCALING DB".PV."FLOW INDICATOR TRANSMITTER 505");
END_REGION

REGION Network 28: FLOW INDICATOR TRANSMITTER 506
   RUNG wire#powerrail
      "FLOW INDICATOR TRANSMITTER_506"("SCALE MIN" := "AI SCALING DB".MIN."FLOW INDICATOR TRANSMITTER 506", "SCALE MAX" := "AI SCALING DB".MAX."FLOW INDICATOR TRANSMITTER 506", INPUT := "FLOW INDICATOR TRANSMITTER 506", "RAW MIN" := 0, "RAW MAX" := 27648, "PV VALUE" => "AI SCALING DB".PV."FLOW INDICATOR TRANSMITTER 506")
   END_RUNG
   // the same network as SCL:
   "FLOW INDICATOR TRANSMITTER_506"("SCALE MIN" := "AI SCALING DB".MIN."FLOW INDICATOR TRANSMITTER 506",   // "SCALE"
                           "SCALE MAX" := "AI SCALING DB".MAX."FLOW INDICATOR TRANSMITTER 506",
                           INPUT := "FLOW INDICATOR TRANSMITTER 506",
                           "RAW MIN" := 0,
                           "RAW MAX" := 27648,
                           "PV VALUE" => "AI SCALING DB".PV."FLOW INDICATOR TRANSMITTER 506");
END_REGION

REGION Network 29: FLOW INDICATOR TRANSMITTER 507
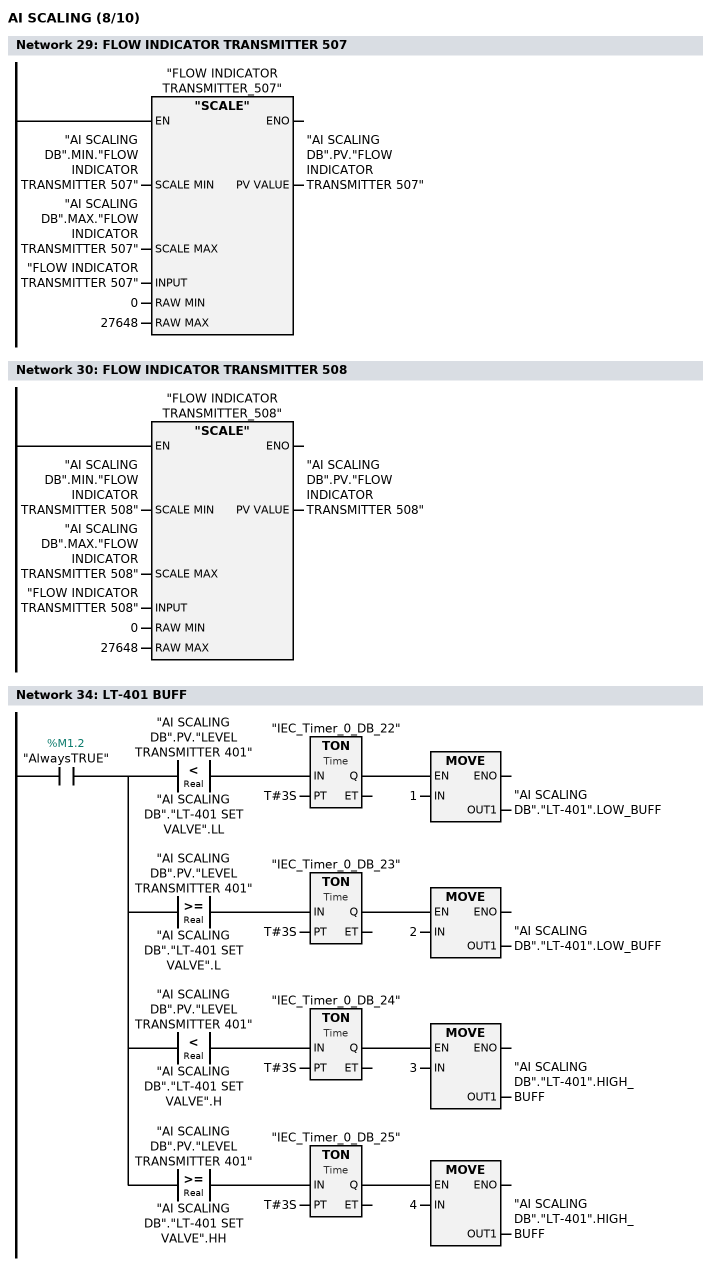
   RUNG wire#powerrail
      "FLOW INDICATOR TRANSMITTER_507"("SCALE MIN" := "AI SCALING DB".MIN."FLOW INDICATOR TRANSMITTER 507", "SCALE MAX" := "AI SCALING DB".MAX."FLOW INDICATOR TRANSMITTER 507", INPUT := "FLOW INDICATOR TRANSMITTER 507", "RAW MIN" := 0, "RAW MAX" := 27648, "PV VALUE" => "AI SCALING DB".PV."FLOW INDICATOR TRANSMITTER 507")
   END_RUNG
   // the same network as SCL:
   "FLOW INDICATOR TRANSMITTER_507"("SCALE MIN" := "AI SCALING DB".MIN."FLOW INDICATOR TRANSMITTER 507",   // "SCALE"
                           "SCALE MAX" := "AI SCALING DB".MAX."FLOW INDICATOR TRANSMITTER 507",
                           INPUT := "FLOW INDICATOR TRANSMITTER 507",
                           "RAW MIN" := 0,
                           "RAW MAX" := 27648,
                           "PV VALUE" => "AI SCALING DB".PV."FLOW INDICATOR TRANSMITTER 507");
END_REGION

REGION Network 30: FLOW INDICATOR TRANSMITTER 508
   RUNG wire#powerrail
      "FLOW INDICATOR TRANSMITTER_508"("SCALE MIN" := "AI SCALING DB".MIN."FLOW INDICATOR TRANSMITTER 508", "SCALE MAX" := "AI SCALING DB".MAX."FLOW INDICATOR TRANSMITTER 508", INPUT := "FLOW INDICATOR TRANSMITTER 508", "RAW MIN" := 0, "RAW MAX" := 27648, "PV VALUE" => "AI SCALING DB".PV."FLOW INDICATOR TRANSMITTER 508")
   END_RUNG
   // the same network as SCL:
   "FLOW INDICATOR TRANSMITTER_508"("SCALE MIN" := "AI SCALING DB".MIN."FLOW INDICATOR TRANSMITTER 508",   // "SCALE"
                           "SCALE MAX" := "AI SCALING DB".MAX."FLOW INDICATOR TRANSMITTER 508",
                           INPUT := "FLOW INDICATOR TRANSMITTER 508",
                           "RAW MIN" := 0,
                           "RAW MAX" := 27648,
                           "PV VALUE" => "AI SCALING DB".PV."FLOW INDICATOR TRANSMITTER 508");
END_REGION

REGION Network 34: LT-401 BUFF
   RUNG wire#powerrail
      Contact( "AlwaysTRUE" )
      wire#w1
      { S7_Templates := "SrcType := Real" } LT_Contact(in1 := "AI SCALING DB".PV."LEVEL TRANSMITTER 401", in2 := "AI SCALING DB"."LT-401 SET VALVE".LL)
      { S7_Templates := "time_type := Time" } "IEC_Timer_0_DB_22".TON(pt := T#3S, et =>)
      Move(in := 1, out1 => "AI SCALING DB"."LT-401".LOW_BUFF)
   END_RUNG
   RUNG wire#w1
      { S7_Templates := "SrcType := Real" } GE_Contact(in1 := "AI SCALING DB".PV."LEVEL TRANSMITTER 401", in2 := "AI SCALING DB"."LT-401 SET VALVE".L)
      { S7_Templates := "time_type := Time" } "IEC_Timer_0_DB_23".TON(pt := T#3S, et =>)
      Move(in := 2, out1 => "AI SCALING DB"."LT-401".LOW_BUFF)
   END_RUNG
   RUNG wire#w1
      { S7_Templates := "SrcType := Real" } LT_Contact(in1 := "AI SCALING DB".PV."LEVEL TRANSMITTER 401", in2 := "AI SCALING DB"."LT-401 SET VALVE".H)
      { S7_Templates := "time_type := Time" } "IEC_Timer_0_DB_24".TON(pt := T#3S, et =>)
      Move(in := 3, out1 => "AI SCALING DB"."LT-401".HIGH_BUFF)
   END_RUNG
   RUNG wire#w1
      { S7_Templates := "SrcType := Real" } GE_Contact(in1 := "AI SCALING DB".PV."LEVEL TRANSMITTER 401", in2 := "AI SCALING DB"."LT-401 SET VALVE".HH)
      { S7_Templates := "time_type := Time" } "IEC_Timer_0_DB_25".TON(pt := T#3S, et =>)
      Move(in := 4, out1 => "AI SCALING DB"."LT-401".HIGH_BUFF)
   END_RUNG
   // the same network as SCL:
   "IEC_Timer_0_DB_22".TON(IN := "AlwaysTRUE" AND ("AI SCALING DB".PV."LEVEL TRANSMITTER 401" < "AI SCALING DB"."LT-401 SET VALVE".LL),
                           PT := T#3S);
   IF "IEC_Timer_0_DB_22".Q THEN "AI SCALING DB"."LT-401".LOW_BUFF := 1; END_IF;
   "IEC_Timer_0_DB_23".TON(IN := "AlwaysTRUE" AND ("AI SCALING DB".PV."LEVEL TRANSMITTER 401" >= "AI SCALING DB"."LT-401 SET VALVE".L),
                           PT := T#3S);
   IF "IEC_Timer_0_DB_23".Q THEN "AI SCALING DB"."LT-401".LOW_BUFF := 2; END_IF;
   "IEC_Timer_0_DB_24".TON(IN := "AlwaysTRUE" AND ("AI SCALING DB".PV."LEVEL TRANSMITTER 401" < "AI SCALING DB"."LT-401 SET VALVE".H),
                           PT := T#3S);
   IF "IEC_Timer_0_DB_24".Q THEN "AI SCALING DB"."LT-401".HIGH_BUFF := 3; END_IF;
   "IEC_Timer_0_DB_25".TON(IN := "AlwaysTRUE" AND ("AI SCALING DB".PV."LEVEL TRANSMITTER 401" >= "AI SCALING DB"."LT-401 SET VALVE".HH),
                           PT := T#3S);
   IF "IEC_Timer_0_DB_25".Q THEN "AI SCALING DB"."LT-401".HIGH_BUFF := 4; END_IF;
END_REGION

REGION Network 35: LT-501 BUFF
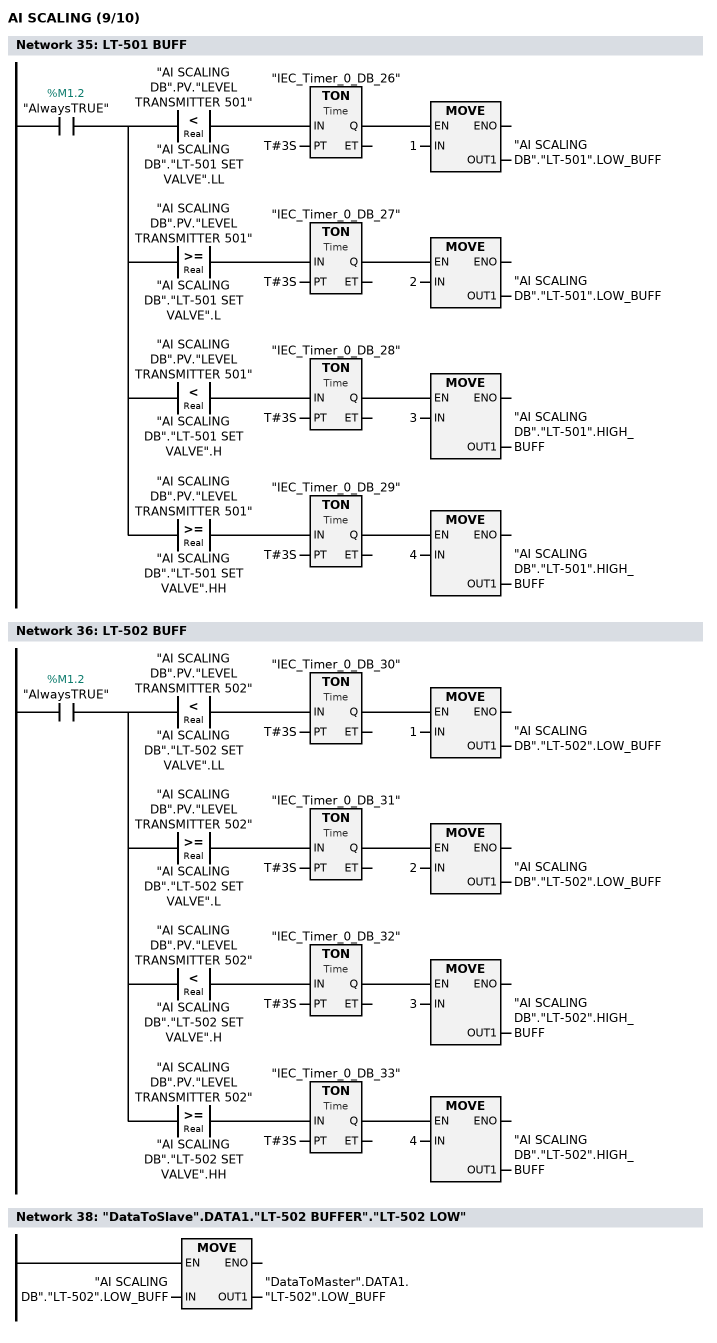
   RUNG wire#powerrail
      Contact( "AlwaysTRUE" )
      wire#w1
      { S7_Templates := "SrcType := Real" } LT_Contact(in1 := "AI SCALING DB".PV."LEVEL TRANSMITTER 501", in2 := "AI SCALING DB"."LT-501 SET VALVE".LL)
      { S7_Templates := "time_type := Time" } "IEC_Timer_0_DB_26".TON(pt := T#3S, et =>)
      Move(in := 1, out1 => "AI SCALING DB"."LT-501".LOW_BUFF)
   END_RUNG
   RUNG wire#w1
      { S7_Templates := "SrcType := Real" } GE_Contact(in1 := "AI SCALING DB".PV."LEVEL TRANSMITTER 501", in2 := "AI SCALING DB"."LT-501 SET VALVE".L)
      { S7_Templates := "time_type := Time" } "IEC_Timer_0_DB_27".TON(pt := T#3S, et =>)
      Move(in := 2, out1 => "AI SCALING DB"."LT-501".LOW_BUFF)
   END_RUNG
   RUNG wire#w1
      { S7_Templates := "SrcType := Real" } LT_Contact(in1 := "AI SCALING DB".PV."LEVEL TRANSMITTER 501", in2 := "AI SCALING DB"."LT-501 SET VALVE".H)
      { S7_Templates := "time_type := Time" } "IEC_Timer_0_DB_28".TON(pt := T#3S, et =>)
      Move(in := 3, out1 => "AI SCALING DB"."LT-501".HIGH_BUFF)
   END_RUNG
   RUNG wire#w1
      { S7_Templates := "SrcType := Real" } GE_Contact(in1 := "AI SCALING DB".PV."LEVEL TRANSMITTER 501", in2 := "AI SCALING DB"."LT-501 SET VALVE".HH)
      { S7_Templates := "time_type := Time" } "IEC_Timer_0_DB_29".TON(pt := T#3S, et =>)
      Move(in := 4, out1 => "AI SCALING DB"."LT-501".HIGH_BUFF)
   END_RUNG
   // the same network as SCL:
   "IEC_Timer_0_DB_26".TON(IN := "AlwaysTRUE" AND ("AI SCALING DB".PV."LEVEL TRANSMITTER 501" < "AI SCALING DB"."LT-501 SET VALVE".LL),
                           PT := T#3S);
   IF "IEC_Timer_0_DB_26".Q THEN "AI SCALING DB"."LT-501".LOW_BUFF := 1; END_IF;
   "IEC_Timer_0_DB_27".TON(IN := "AlwaysTRUE" AND ("AI SCALING DB".PV."LEVEL TRANSMITTER 501" >= "AI SCALING DB"."LT-501 SET VALVE".L),
                           PT := T#3S);
   IF "IEC_Timer_0_DB_27".Q THEN "AI SCALING DB"."LT-501".LOW_BUFF := 2; END_IF;
   "IEC_Timer_0_DB_28".TON(IN := "AlwaysTRUE" AND ("AI SCALING DB".PV."LEVEL TRANSMITTER 501" < "AI SCALING DB"."LT-501 SET VALVE".H),
                           PT := T#3S);
   IF "IEC_Timer_0_DB_28".Q THEN "AI SCALING DB"."LT-501".HIGH_BUFF := 3; END_IF;
   "IEC_Timer_0_DB_29".TON(IN := "AlwaysTRUE" AND ("AI SCALING DB".PV."LEVEL TRANSMITTER 501" >= "AI SCALING DB"."LT-501 SET VALVE".HH),
                           PT := T#3S);
   IF "IEC_Timer_0_DB_29".Q THEN "AI SCALING DB"."LT-501".HIGH_BUFF := 4; END_IF;
END_REGION

